LIN {X 0,Y 281.537,Z 487.928,A -85,B 0,C 180,E1 -17516.689,E2 -17516.689} C_VEL
LIN {X 0,Y 281.333,Z 491.576,A -85,B 0,C 180,E1 -17518.052,E2 -17518.052} C_VEL
LIN {X 0,Y 285.942,Z 506.962,A -85,B 0,C 180,E1 -17519.189,E2 -17519.189} C_VEL
LIN {X 0,Y 289.242,Z 521.138,A -85,B 0,C 180,E1 -17520.411,E2 -17520.411} C_VEL
LIN {X 0,Y 291.221,Z 533.956,A -85,B 0,C 180,E1 -17521.672,E2 -17521.672} C_VEL
LIN {X 0,Y 291.985,Z 542.885,A -85,B 0,C 180,E1 -17522.647,E2 -17522.647} C_VEL
LIN {X 0,Y 290.191,Z 554.779,A -85,B 0,C 180,E1 -17523.912,E2 -17523.912} C_VEL
LIN {X 0,Y 287.889,Z 566.73,A -85,B 0,C 180,E1 -17525.48,E2 -17525.48} C_VEL
LIN {X 0,Y 285.539,Z 577.345,A -85,B 0,C 180,E1 -17527.191,E2 -17527.191} C_VEL
LIN {X 0,Y 283.172,Z 587.851,A -85,B 0,C 180,E1 -17529.288,E2 -17529.288} C_VEL
LIN {X 0,Y 281.044,Z 596.524,A -85,B 0,C 180,E1 -17531.408,E2 -17531.408} C_VEL
LIN {X 0,Y 279.492,Z 603.728,A -85,B 0,C 180,E1 -17533.567,E2 -17533.567} C_VEL
LIN {X 0,Y 277.872,Z 610.612,A -85,B 0,C 180,E1 -17536.097,E2 -17536.097} C_VEL
LIN {X 0,Y 276.558,Z 616.782,A -85,B 0,C 180,E1 -17539.013,E2 -17539.013} C_VEL
LIN {X 0,Y 275.927,Z 620.289,A -85,B 0,C 180,E1 -17541.209,E2 -17541.209} C_VEL
LIN {X 0,Y 275.417,Z 623.71,A -85,B 0,C 180,E1 -17544.142,E2 -17544.142} C_VEL
LIN {X 0,Y 275.26,Z 625.741,A -85,B 0,C 180,E1 -17547.073,E2 -17547.073} C_VEL
LIN {X 0,Y 275.22,Z 626.437,A -85,B 0,C 180,E1 -17550,E2 -17550} C_VEL
LIN {X 0,Y 275.258,Z 625.8,A -85,B 0,C 180,E1 -17552.927,E2 -17552.927} C_VEL
LIN {X 0,Y 275.416,Z 623.816,A -85,B 0,C 180,E1 -17555.858,E2 -17555.858} C_VEL
LIN {X 0,Y 275.925,Z 620.448,A -85,B 0,C 180,E1 -17558.791,E2 -17558.791} C_VEL
LIN {X 0,Y 276.784,Z 615.594,A -85,B 0,C 180,E1 -17561.72,E2 -17561.72} C_VEL
LIN {X 0,Y 277.821,Z 610.887,A -85,B 0,C 180,E1 -17563.905,E2 -17563.905} C_VEL
LIN {X 0,Y 279.41,Z 604.105,A -85,B 0,C 180,E1 -17566.423,E2 -17566.423} C_VEL
LIN {X 0,Y 281.359,Z 595.594,A -85,B 0,C 180,E1 -17568.949,E2 -17568.949} C_VEL
LIN {X 0,Y 283.505,Z 586.735,A -85,B 0,C 180,E1 -17571.067,E2 -17571.067} C_VEL
LIN {X 0,Y 285.86,Z 576.009,A -85,B 0,C 180,E1 -17573.164,E2 -17573.164} C_VEL
LIN {X 0,Y 288.304,Z 565.121,A -85,B 0,C 180,E1 -17574.866,E2 -17574.866} C_VEL
LIN {X 0,Y 290.592,Z 552.488,A -85,B 0,C 180,E1 -17576.467,E2 -17576.467} C_VEL
LIN {X 0,Y 292.06,Z 542.514,A -85,B 0,C 180,E1 -17577.505,E2 -17577.505} C_VEL
LIN {X 0,Y 290.791,Z 530.649,A -85,B 0,C 180,E1 -17578.792,E2 -17578.792} C_VEL
LIN {X 0,Y 288.442,Z 517.113,A -85,B 0,C 180,E1 -17580.077,E2 -17580.077} C_VEL
LIN {X 0,Y 284.962,Z 503.246,A -85,B 0,C 180,E1 -17581.223,E2 -17581.223} C_VEL
LIN {X 0,Y 281.275,Z 491.314,A -85,B 0,C 180,E1 -17582.094,E2 -17582.094} C_VEL
LIN {X 0,Y 282.191,Z 480.989,A -85,B 0,C 180,E1 -17586.263,E2 -17586.263} C_VEL
LIN {X 0,Y 283.218,Z 471.628,A -85,B 0,C 180,E1 -17590.18,E2 -17590.18} C_VEL
LIN {X 0,Y 283.249,Z 467.404,A -85,B 0,C 180,E1 -17592.061,E2 -17592.061} C_VEL
LIN {X 0,Y 281.982,Z 459.837,A -85,B 0,C 180,E1 -17595.744,E2 -17595.744} C_VEL
LIN {X 0,Y 280.547,Z 452.755,A -85,B 0,C 180,E1 -17599.358,E2 -17599.358} C_VEL
LIN {X 0,Y 279.094,Z 446.242,A -85,B 0,C 180,E1 -17602.817,E2 -17602.817} C_VEL
LIN {X 0,Y 277.267,Z 439.563,A -85,B 0,C 180,E1 -17606.638,E2 -17606.638} C_VEL
LIN {X 0,Y 277.277,Z 439.557,A -85,B 0,C 180,E1 -17609.73,E2 -17609.73} C_VEL
LIN {X 0,Y 282.338,Z 455.073,A -85,B 0,C 180,E1 -17611.505,E2 -17611.505} C_VEL
LIN {X 0,Y 286.61,Z 469.194,A -85,B 0,C 180,E1 -17613.343,E2 -17613.343} C_VEL
LIN {X 0,Y 287.766,Z 473.23,A -85,B 0,C 180,E1 -17613.921,E2 -17613.921} C_VEL
LIN {X 0,Y 286.168,Z 485.511,A -85,B 0,C 180,E1 -17615.516,E2 -17615.516} C_VEL
LIN {X 0,Y 284.267,Z 498.156,A -85,B 0,C 180,E1 -17617.467,E2 -17617.467} C_VEL
LIN {X 0,Y 282.497,Z 509.782,A -85,B 0,C 180,E1 -17619.617,E2 -17619.617} C_VEL
LIN {X 0,Y 280.89,Z 519.521,A -85,B 0,C 180,E1 -17621.752,E2 -17621.752} C_VEL
LIN {X 0,Y 279.534,Z 529.33,A -85,B 0,C 180,E1 -17624.319,E2 -17624.319} C_VEL
LIN {X 0,Y 279.286,Z 530.981,A -85,B 0,C 180,E1 -17624.798,E2 -17624.798} C_VEL
LIN {X 0,Y 278.057,Z 534.299,A -85,B 0,C 180,E1 -17625.786,E2 -17625.786} C_VEL
LIN {X 0,Y 274.501,Z 539.379,A -85,B 0,C 180,E1 -17627.397,E2 -17627.397} C_VEL
LIN {X 0,Y 271.128,Z 544.003,A -85,B 0,C 180,E1 -17629.093,E2 -17629.093} C_VEL
LIN {X 0,Y 270.198,Z 546.576,A -85,B 0,C 180,E1 -17630.195,E2 -17630.195} C_VEL
LIN {X 0,Y 269.657,Z 552.512,A -85,B 0,C 180,E1 -17633.265,E2 -17633.265} C_VEL
LIN {X 0,Y 269.565,Z 555.917,A -85,B 0,C 180,E1 -17635.514,E2 -17635.514} C_VEL
LIN {X 0,Y 269.279,Z 559.358,A -85,B 0,C 180,E1 -17638.504,E2 -17638.504} C_VEL
LIN {X 0,Y 269.373,Z 561.559,A -85,B 0,C 180,E1 -17641.495,E2 -17641.495} C_VEL
LIN {X 0,Y 269.987,Z 562.568,A -85,B 0,C 180,E1 -17644.479,E2 -17644.479} C_VEL
LIN {X 0,Y 271.059,Z 562.393,A -85,B 0,C 180,E1 -17647.449,E2 -17647.449} C_VEL
LIN {X 0,Y 272.422,Z 561.092,A -85,B 0,C 180,E1 -17650.404,E2 -17650.404} C_VEL
LIN {X 0,Y 274.151,Z 558.636,A -85,B 0,C 180,E1 -17653.339,E2 -17653.339} C_VEL
LIN {X 0,Y 276.346,Z 555.017,A -85,B 0,C 180,E1 -17656.245,E2 -17656.245} C_VEL
LIN {X 0,Y 279.276,Z 550.056,A -85,B 0,C 180,E1 -17659.096,E2 -17659.096} C_VEL
LIN {X 0,Y 281.817,Z 545.44,A -85,B 0,C 180,E1 -17661.199,E2 -17661.199} C_VEL
LIN {X 0,Y 286.188,Z 537.267,A -85,B 0,C 180,E1 -17664.197,E2 -17664.197} C_VEL
LIN {X 0,Y 290.835,Z 527.733,A -85,B 0,C 180,E1 -17666.942,E2 -17666.942} C_VEL
LIN {X 0,Y 295.354,Z 517.993,A -85,B 0,C 180,E1 -17669.196,E2 -17669.196} C_VEL
LIN {X 0,Y 299.707,Z 508.242,A -85,B 0,C 180,E1 -17671.057,E2 -17671.057} C_VEL
LIN {X 0,Y 303.199,Z 499.743,A -85,B 0,C 180,E1 -17672.464,E2 -17672.464} C_VEL
LIN {X 0,Y 303.462,Z 498.058,A -85,B 0,C 180,E1 -17672.86,E2 -17672.86} C_VEL
LIN {X 0,Y 302.842,Z 492.133,A -85,B 0,C 180,E1 -17674.941,E2 -17674.941} C_VEL
LIN {X 0,Y 302.211,Z 488.957,A -85,B 0,C 180,E1 -17676.323,E2 -17676.323} C_VEL
LIN {X 0,Y 301.253,Z 487.359,A -85,B 0,C 180,E1 -17677.515,E2 -17677.515} C_VEL
LIN {X 0,Y 299.735,Z 486.025,A -85,B 0,C 180,E1 -17679.307,E2 -17679.307} C_VEL
LIN {X 0,Y 298.35,Z 485.722,A -85,B 0,C 180,E1 -17681.267,E2 -17681.267} C_VEL
LIN {X 0,Y 297.068,Z 486.886,A -85,B 0,C 180,E1 -17683.32,E2 -17683.32} C_VEL
LIN {X 0,Y 296.328,Z 488.596,A -85,B 0,C 180,E1 -17684.642,E2 -17684.642} C_VEL
LIN {X 0,Y 294.815,Z 495.196,A -85,B 0,C 180,E1 -17687.646,E2 -17687.646} C_VEL
LIN {X 0,Y 294.665,Z 498.561,A -85,B 0,C 180,E1 -17689.057,E2 -17689.057} C_VEL
LIN {X 0,Y 294.316,Z 505.488,A -85,B 0,C 180,E1 -17691.235,E2 -17691.235} C_VEL
LIN {X 0,Y 294.003,Z 512.7,A -85,B 0,C 180,E1 -17693.139,E2 -17693.139} C_VEL
LIN {X 0,Y 293.508,Z 520.438,A -85,B 0,C 180,E1 -17694.923,E2 -17694.923} C_VEL
LIN {X 0,Y 292.34,Z 530.113,A -85,B 0,C 180,E1 -17696.885,E2 -17696.885} C_VEL
LIN {X 0,Y 290.404,Z 539.351,A -85,B 0,C 180,E1 -17698.604,E2 -17698.604} C_VEL
LIN {X 0,Y 287.008,Z 552.38,A -85,B 0,C 180,E1 -17701.078,E2 -17701.078} C_VEL
LIN {X 0,Y 285.923,Z 557.42,A -85,B 0,C 180,E1 -17702.159,E2 -17702.159} C_VEL
LIN {X 0,Y 282.042,Z 567.163,A -85,B 0,C 180,E1 -17704.147,E2 -17704.147} C_VEL
LIN {X 0,Y 281.188,Z 569.389,A -85,B 0,C 180,E1 -17704.658,E2 -17704.658} C_VEL
LIN {X 0,Y 278.988,Z 579.397,A -85,B 0,C 180,E1 -17706.231,E2 -17706.231} C_VEL
LIN {X 0,Y 276.824,Z 588.72,A -85,B 0,C 180,E1 -17708.008,E2 -17708.008} C_VEL
LIN {X 0,Y 274.587,Z 598.075,A -85,B 0,C 180,E1 -17710.176,E2 -17710.176} C_VEL
LIN {X 0,Y 272.687,Z 606.145,A -85,B 0,C 180,E1 -17712.479,E2 -17712.479} C_VEL
LIN {X 0,Y 271.131,Z 613.215,A -85,B 0,C 180,E1 -17714.977,E2 -17714.977} C_VEL
LIN {X 0,Y 269.555,Z 619.823,A -85,B 0,C 180,E1 -17717.961,E2 -17717.961} C_VEL
LIN {X 0,Y 268.738,Z 624.77,A -85,B 0,C 180,E1 -17720.972,E2 -17720.972} C_VEL
LIN {X 0,Y 268.305,Z 628.21,A -85,B 0,C 180,E1 -17723.986,E2 -17723.986} C_VEL
LIN {X 0,Y 268.201,Z 630.245,A -85,B 0,C 180,E1 -17726.996,E2 -17726.996} C_VEL
LIN {X 0,Y 268.193,Z 630.919,A -85,B 0,C 180,E1 -17730,E2 -17730} C_VEL
LIN {X 0,Y 268.199,Z 630.236,A -85,B 0,C 180,E1 -17733.004,E2 -17733.004} C_VEL
LIN {X 0,Y 268.299,Z 628.194,A -85,B 0,C 180,E1 -17736.014,E2 -17736.014} C_VEL
LIN {X 0,Y 268.714,Z 624.745,A -85,B 0,C 180,E1 -17739.028,E2 -17739.028} C_VEL
LIN {X 0,Y 269.537,Z 619.783,A -85,B 0,C 180,E1 -17742.04,E2 -17742.04} C_VEL
LIN {X 0,Y 271.095,Z 613.165,A -85,B 0,C 180,E1 -17745.025,E2 -17745.025} C_VEL
LIN {X 0,Y 272.585,Z 606.058,A -85,B 0,C 180,E1 -17747.535,E2 -17747.535} C_VEL
LIN {X 0,Y 274.558,Z 597.994,A -85,B 0,C 180,E1 -17749.826,E2 -17749.826} C_VEL
LIN {X 0,Y 276.769,Z 588.618,A -85,B 0,C 180,E1 -17751.996,E2 -17751.996} C_VEL
LIN {X 0,Y 279.183,Z 578.215,A -85,B 0,C 180,E1 -17753.949,E2 -17753.949} C_VEL
LIN {X 0,Y 281.738,Z 566.352,A -85,B 0,C 180,E1 -17755.741,E2 -17755.741} C_VEL
LIN {X 0,Y 283.764,Z 553.932,A -85,B 0,C 180,E1 -17757.27,E2 -17757.27} C_VEL
LIN {X 0,Y 283.178,Z 541.327,A -85,B 0,C 180,E1 -17758.748,E2 -17758.748} C_VEL
LIN {X 0,Y 281.859,Z 528.409,A -85,B 0,C 180,E1 -17760.039,E2 -17760.039} C_VEL
LIN {X 0,Y 280.013,Z 514.186,A -85,B 0,C 180,E1 -17761.189,E2 -17761.189} C_VEL
LIN {X 0,Y 277.183,Z 503.097,A -85,B 0,C 180,E1 -17762.029,E2 -17762.029} C_VEL
LIN {X 0,Y 272.899,Z 489.832,A -85,B 0,C 180,E1 -17763.066,E2 -17763.066} C_VEL
LIN {X 0,Y 271.754,Z 479.976,A -85,B 0,C 180,E1 -17765.129,E2 -17765.129} C_VEL
LIN {X 0,Y 270.998,Z 474.249,A -85,B 0,C 180,E1 -17766.39,E2 -17766.39} C_VEL
LIN {X 0,Y 271.661,Z 468.446,A -85,B 0,C 180,E1 -17770.298,E2 -17770.298} C_VEL
LIN {X 0,Y 272.367,Z 462.83,A -85,B 0,C 180,E1 -17774.162,E2 -17774.162} C_VEL
LIN {X 0,Y 272.893,Z 458.634,A -85,B 0,C 180,E1 -17777.089,E2 -17777.089} C_VEL
LIN {X 0,Y 272.752,Z 454.791,A -85,B 0,C 180,E1 -17779.896,E2 -17779.896} C_VEL
LIN {X 0,Y 271.911,Z 450.029,A -85,B 0,C 180,E1 -17783.525,E2 -17783.525} C_VEL
LIN {X 0,Y 271.032,Z 444.568,A -85,B 0,C 180,E1 -17787.888,E2 -17787.888} C_VEL
LIN {X 0,Y 270.308,Z 440.441,A -85,B 0,C 180,E1 -17791.462,E2 -17791.462} C_VEL
LIN {X 0,Y 270.278,Z 440.435,A -85,B 0,C 180,E1 -17795.519,E2 -17795.519} C_VEL
LIN {X 0,Y 270.303,Z 440.421,A -85,B 0,C 180,E1 -17800.245,E2 -17800.245} C_VEL
LIN {X 0,Y 270.404,Z 440.405,A -85,B 0,C 180,E1 -17804.936,E2 -17804.936} C_VEL
LIN {X 0,Y 270.411,Z 440.415,A -85,B 0,C 180,E1 -17809.518,E2 -17809.518} C_VEL
LIN {X 0,Y 270.582,Z 440.392,A -85,B 0,C 180,E1 -17812.538,E2 -17812.538} C_VEL
LIN {X 0,Y 270.789,Z 440.366,A -85,B 0,C 180,E1 -17818.513,E2 -17818.513} C_VEL
LIN {X 0,Y 270.789,Z 440.369,A -85,B 0,C 180,E1 -17821.487,E2 -17821.487} C_VEL
LIN {X 0,Y 270.613,Z 440.387,A -85,B 0,C 180,E1 -17827.461,E2 -17827.461} C_VEL
LIN {X 0,Y 270.444,Z 440.419,A -85,B 0,C 180,E1 -17830.481,E2 -17830.481} C_VEL
LIN {X 0,Y 270.405,Z 440.418,A -85,B 0,C 180,E1 -17835.065,E2 -17835.065} C_VEL
LIN {X 0,Y 270.301,Z 440.432,A -85,B 0,C 180,E1 -17839.756,E2 -17839.756} C_VEL
LIN {X 0,Y 270.239,Z 440.448,A -85,B 0,C 180,E1 -17844.589,E2 -17844.589} C_VEL
LIN {X 0,Y 270.273,Z 440.44,A -85,B 0,C 180,E1 -17847.909,E2 -17847.909} C_VEL
LIN {X 0,Y 270.237,Z 440.596,A -85,B 0,C 180,E1 -17852.438,E2 -17852.438} C_VEL
LIN {X 0,Y 271.699,Z 445.957,A -85,B 0,C 180,E1 -17855.592,E2 -17855.592} C_VEL
LIN {X 0,Y 273.306,Z 452.497,A -85,B 0,C 180,E1 -17859.194,E2 -17859.194} C_VEL
LIN {X 0,Y 274.734,Z 459,A -85,B 0,C 180,E1 -17862.679,E2 -17862.679} C_VEL
LIN {X 0,Y 276.105,Z 466.777,A -85,B 0,C 180,E1 -17866.586,E2 -17866.586} C_VEL
LIN {X 0,Y 276.618,Z 471.079,A -85,B 0,C 180,E1 -17868.656,E2 -17868.656} C_VEL
LIN {X 0,Y 275.952,Z 477.382,A -85,B 0,C 180,E1 -17871.394,E2 -17871.394} C_VEL
LIN {X 0,Y 274.979,Z 486.758,A -85,B 0,C 180,E1 -17875.306,E2 -17875.306} C_VEL
LIN {X 0,Y 274.573,Z 491.348,A -85,B 0,C 180,E1 -17877.163,E2 -17877.163} C_VEL
LIN {X 0,Y 279.426,Z 507.204,A -85,B 0,C 180,E1 -17878.401,E2 -17878.401} C_VEL
LIN {X 0,Y 282.623,Z 521.049,A -85,B 0,C 180,E1 -17879.638,E2 -17879.638} C_VEL
LIN {X 0,Y 284.651,Z 533.995,A -85,B 0,C 180,E1 -17880.956,E2 -17880.956} C_VEL
LIN {X 0,Y 285.511,Z 544.157,A -85,B 0,C 180,E1 -17882.115,E2 -17882.115} C_VEL
LIN {X 0,Y 283.482,Z 556.585,A -85,B 0,C 180,E1 -17883.497,E2 -17883.497} C_VEL
LIN {X 0,Y 281.179,Z 567.932,A -85,B 0,C 180,E1 -17885.053,E2 -17885.053} C_VEL
LIN {X 0,Y 278.967,Z 577.399,A -85,B 0,C 180,E1 -17886.622,E2 -17886.622} C_VEL
LIN {X 0,Y 276.535,Z 587.906,A -85,B 0,C 180,E1 -17888.767,E2 -17888.767} C_VEL
LIN {X 0,Y 274.293,Z 596.579,A -85,B 0,C 180,E1 -17890.932,E2 -17890.932} C_VEL
LIN {X 0,Y 272.609,Z 603.855,A -85,B 0,C 180,E1 -17893.164,E2 -17893.164} C_VEL
LIN {X 0,Y 271.448,Z 608.885,A -85,B 0,C 180,E1 -17894.995,E2 -17894.995} C_VEL
LIN {X 0,Y 270.171,Z 613.968,A -85,B 0,C 180,E1 -17897.226,E2 -17897.226} C_VEL
LIN {X 0,Y 269.072,Z 619.296,A -85,B 0,C 180,E1 -17900.225,E2 -17900.225} C_VEL
LIN {X 0,Y 268.56,Z 622.238,A -85,B 0,C 180,E1 -17902.482,E2 -17902.482} C_VEL
LIN {X 0,Y 268.203,Z 624.954,A -85,B 0,C 180,E1 -17905.491,E2 -17905.491} C_VEL
LIN {X 0,Y 268.141,Z 626.313,A -85,B 0,C 180,E1 -17908.498,E2 -17908.498} C_VEL
LIN {X 0,Y 268.14,Z 626.344,A -85,B 0,C 180,E1 -17911.502,E2 -17911.502} C_VEL
LIN {X 0,Y 268.198,Z 625.035,A -85,B 0,C 180,E1 -17914.509,E2 -17914.509} C_VEL
LIN {X 0,Y 268.549,Z 622.368,A -85,B 0,C 180,E1 -17917.519,E2 -17917.519} C_VEL
LIN {X 0,Y 269.276,Z 618.272,A -85,B 0,C 180,E1 -17920.527,E2 -17920.527} C_VEL
LIN {X 0,Y 270.443,Z 612.62,A -85,B 0,C 180,E1 -17923.526,E2 -17923.526} C_VEL
LIN {X 0,Y 272.169,Z 606.227,A -85,B 0,C 180,E1 -17926.116,E2 -17926.116} C_VEL
LIN {X 0,Y 273.991,Z 598.286,A -85,B 0,C 180,E1 -17928.701,E2 -17928.701} C_VEL
LIN {X 0,Y 276.058,Z 589.958,A -85,B 0,C 180,E1 -17930.88,E2 -17930.88} C_VEL
LIN {X 0,Y 278.468,Z 579.891,A -85,B 0,C 180,E1 -17933.029,E2 -17933.029} C_VEL
LIN {X 0,Y 281.049,Z 568.621,A -85,B 0,C 180,E1 -17934.96,E2 -17934.96} C_VEL
LIN {X 0,Y 283.378,Z 557.414,A -85,B 0,C 180,E1 -17936.514,E2 -17936.514} C_VEL
LIN {X 0,Y 285.598,Z 543.959,A -85,B 0,C 180,E1 -17938.017,E2 -17938.017} C_VEL
LIN {X 0,Y 284.481,Z 532.457,A -85,B 0,C 180,E1 -17939.326,E2 -17939.326} C_VEL
LIN {X 0,Y 282.182,Z 518.597,A -85,B 0,C 180,E1 -17940.71,E2 -17940.71} C_VEL
LIN {X 0,Y 279.027,Z 505.702,A -85,B 0,C 180,E1 -17941.847,E2 -17941.847} C_VEL
LIN {X 0,Y 274.583,Z 491.242,A -85,B 0,C 180,E1 -17943.003,E2 -17943.003} C_VEL
LIN {X 0,Y 275.604,Z 480.868,A -85,B 0,C 180,E1 -17947.274,E2 -17947.274} C_VEL
LIN {X 0,Y 276.534,Z 472.831,A -85,B 0,C 180,E1 -17950.697,E2 -17950.697} C_VEL
LIN {X 0,Y 276.43,Z 468.936,A -85,B 0,C 180,E1 -17952.498,E2 -17952.498} C_VEL
LIN {X 0,Y 275.429,Z 462.706,A -85,B 0,C 180,E1 -17955.599,E2 -17955.599} C_VEL
LIN {X 0,Y 274.056,Z 455.847,A -85,B 0,C 180,E1 -17959.161,E2 -17959.161} C_VEL
LIN {X 0,Y 272.431,Z 448.564,A -85,B 0,C 180,E1 -17963.103,E2 -17963.103} C_VEL
LIN {X 0,Y 270.575,Z 441.975,A -85,B 0,C 180,E1 -17966.944,E2 -17966.944} C_VEL
LIN {X 0,Y 270.198,Z 440.454,A -85,B 0,C 180,E1 -17967.887,E2 -17967.887} C_VEL
LIN {X 0,Y 270.208,Z 440.438,A -85,B 0,C 180,E1 -17969.262,E2 -17969.262} C_VEL
LIN {X 0,Y 274.919,Z 454.754,A -85,B 0,C 180,E1 -17970.941,E2 -17970.941} C_VEL
LIN {X 0,Y 278.914,Z 467.876,A -85,B 0,C 180,E1 -17972.678,E2 -17972.678} C_VEL
LIN {X 0,Y 280.801,Z 474.405,A -85,B 0,C 180,E1 -17973.624,E2 -17973.624} C_VEL
LIN {X 0,Y 280.034,Z 481.499,A -85,B 0,C 180,E1 -17974.546,E2 -17974.546} C_VEL
LIN {X 0,Y 277.986,Z 494.946,A -85,B 0,C 180,E1 -17976.535,E2 -17976.535} C_VEL
LIN {X 0,Y 276.04,Z 507.187,A -85,B 0,C 180,E1 -17978.727,E2 -17978.727} C_VEL
LIN {X 0,Y 274.271,Z 517.708,A -85,B 0,C 180,E1 -17980.969,E2 -17980.969} C_VEL
LIN {X 0,Y 272.99,Z 526.414,A -85,B 0,C 180,E1 -17983.164,E2 -17983.164} C_VEL
LIN {X 0,Y 271.638,Z 535.137,A -85,B 0,C 180,E1 -17985.771,E2 -17985.771} C_VEL
LIN {X 0,Y 270.592,Z 543.292,A -85,B 0,C 180,E1 -17988.767,E2 -17988.767} C_VEL
LIN {X 0,Y 270.198,Z 546.576,A -85,B 0,C 180,E1 -17990.195,E2 -17990.195} C_VEL
LIN {X 0,Y 269.313,Z 549.046,A -85,B 0,C 180,E1 -17991.317,E2 -17991.317} C_VEL
LIN {X 0,Y 266.197,Z 552.693,A -85,B 0,C 180,E1 -17993.173,E2 -17993.173} C_VEL
LIN {X 0,Y 263.622,Z 555.289,A -85,B 0,C 180,E1 -17994.712,E2 -17994.712} C_VEL
LIN {X 0,Y 262.475,Z 557.024,A -85,B 0,C 180,E1 -17995.927,E2 -17995.927} C_VEL
LIN {X 0,Y 262.353,Z 557.506,A -85,B 0,C 180,E1 -17996.342,E2 -17996.342} C_VEL
LIN {X 0,Y 262.213,Z 559.894,A -85,B 0,C 180,E1 -17998.464,E2 -17998.464} C_VEL
LIN {X 0,Y 262.337,Z 562.272,A -85,B 0,C 180,E1 -18001.535,E2 -18001.535} C_VEL
LIN {X 0,Y 262.976,Z 563.458,A -85,B 0,C 180,E1 -18004.598,E2 -18004.598} C_VEL
LIN {X 0,Y 264.1,Z 563.469,A -85,B 0,C 180,E1 -18007.646,E2 -18007.646} C_VEL
LIN {X 0,Y 265.553,Z 562.332,A -85,B 0,C 180,E1 -18010.676,E2 -18010.676} C_VEL
LIN {X 0,Y 267.384,Z 560.076,A -85,B 0,C 180,E1 -18013.683,E2 -18013.683} C_VEL
LIN {X 0,Y 269.739,Z 556.631,A -85,B 0,C 180,E1 -18016.655,E2 -18016.655} C_VEL
LIN {X 0,Y 272.825,Z 551.933,A -85,B 0,C 180,E1 -18019.565,E2 -18019.565} C_VEL
LIN {X 0,Y 276.545,Z 545.91,A -85,B 0,C 180,E1 -18022.408,E2 -18022.408} C_VEL
LIN {X 0,Y 280.84,Z 538.447,A -85,B 0,C 180,E1 -18025.177,E2 -18025.177} C_VEL
LIN {X 0,Y 284.893,Z 530.882,A -85,B 0,C 180,E1 -18027.471,E2 -18027.471} C_VEL
LIN {X 0,Y 289.778,Z 521.41,A -85,B 0,C 180,E1 -18029.814,E2 -18029.814} C_VEL
LIN {X 0,Y 295.091,Z 510.429,A -85,B 0,C 180,E1 -18032,E2 -18032} C_VEL
LIN {X 0,Y 298.137,Z 503.586,A -85,B 0,C 180,E1 -18033.177,E2 -18033.177} C_VEL
LIN {X 0,Y 298.598,Z 502.215,A -85,B 0,C 180,E1 -18033.465,E2 -18033.465} C_VEL
LIN {X 0,Y 298.353,Z 496.969,A -85,B 0,C 180,E1 -18035.455,E2 -18035.455} C_VEL
LIN {X 0,Y 297.962,Z 494.409,A -85,B 0,C 180,E1 -18036.683,E2 -18036.683} C_VEL
LIN {X 0,Y 296.547,Z 492.579,A -85,B 0,C 180,E1 -18038.548,E2 -18038.548} C_VEL
LIN {X 0,Y 295.293,Z 491.93,A -85,B 0,C 180,E1 -18040.394,E2 -18040.394} C_VEL
LIN {X 0,Y 294.158,Z 492.361,A -85,B 0,C 180,E1 -18042.213,E2 -18042.213} C_VEL
LIN {X 0,Y 292.969,Z 494.251,A -85,B 0,C 180,E1 -18044.081,E2 -18044.081} C_VEL
LIN {X 0,Y 291.354,Z 498.927,A -85,B 0,C 180,E1 -18046.357,E2 -18046.357} C_VEL
LIN {X 0,Y 290.675,Z 503.868,A -85,B 0,C 180,E1 -18048.549,E2 -18048.549} C_VEL
LIN {X 0,Y 289.863,Z 511.203,A -85,B 0,C 180,E1 -18050.921,E2 -18050.921} C_VEL
LIN {X 0,Y 289.105,Z 518.87,A -85,B 0,C 180,E1 -18053.005,E2 -18053.005} C_VEL
LIN {X 0,Y 288.002,Z 527.223,A -85,B 0,C 180,E1 -18054.952,E2 -18054.952} C_VEL
LIN {X 0,Y 286.309,Z 535.869,A -85,B 0,C 180,E1 -18056.751,E2 -18056.751} C_VEL
LIN {X 0,Y 283.557,Z 545.561,A -85,B 0,C 180,E1 -18058.635,E2 -18058.635} C_VEL
LIN {X 0,Y 280.576,Z 555.757,A -85,B 0,C 180,E1 -18060.762,E2 -18060.762} C_VEL
LIN {X 0,Y 279.796,Z 558.934,A -85,B 0,C 180,E1 -18061.494,E2 -18061.494} C_VEL
LIN {X 0,Y 275.141,Z 569.677,A -85,B 0,C 180,E1 -18063.856,E2 -18063.856} C_VEL
LIN {X 0,Y 274.123,Z 572.267,A -85,B 0,C 180,E1 -18064.466,E2 -18064.466} C_VEL
LIN {X 0,Y 271.54,Z 583.248,A -85,B 0,C 180,E1 -18066.349,E2 -18066.349} C_VEL
LIN {X 0,Y 269.025,Z 593.574,A -85,B 0,C 180,E1 -18068.547,E2 -18068.547} C_VEL
LIN {X 0,Y 266.837,Z 602.075,A -85,B 0,C 180,E1 -18070.778,E2 -18070.778} C_VEL
LIN {X 0,Y 264.918,Z 610.174,A -85,B 0,C 180,E1 -18073.43,E2 -18073.43} C_VEL
LIN {X 0,Y 263.335,Z 616.682,A -85,B 0,C 180,E1 -18076.102,E2 -18076.102} C_VEL
LIN {X 0,Y 262.073,Z 622.437,A -85,B 0,C 180,E1 -18079.18,E2 -18079.18} C_VEL
LIN {X 0,Y 261.4,Z 626.613,A -85,B 0,C 180,E1 -18082.274,E2 -18082.274} C_VEL
LIN {X 0,Y 261.105,Z 629.34,A -85,B 0,C 180,E1 -18085.368,E2 -18085.368} C_VEL
LIN {X 0,Y 261.115,Z 630.694,A -85,B 0,C 180,E1 -18088.458,E2 -18088.458} C_VEL
LIN {X 0,Y 261.114,Z 630.689,A -85,B 0,C 180,E1 -18091.542,E2 -18091.542} C_VEL
LIN {X 0,Y 261.1,Z 629.328,A -85,B 0,C 180,E1 -18094.632,E2 -18094.632} C_VEL
LIN {X 0,Y 261.374,Z 626.592,A -85,B 0,C 180,E1 -18097.726,E2 -18097.726} C_VEL
LIN {X 0,Y 262.062,Z 622.402,A -85,B 0,C 180,E1 -18100.82,E2 -18100.82} C_VEL
LIN {X 0,Y 263.318,Z 616.634,A -85,B 0,C 180,E1 -18103.899,E2 -18103.899} C_VEL
LIN {X 0,Y 264.855,Z 610.115,A -85,B 0,C 180,E1 -18106.574,E2 -18106.574} C_VEL
LIN {X 0,Y 266.801,Z 601.997,A -85,B 0,C 180,E1 -18109.225,E2 -18109.225} C_VEL
LIN {X 0,Y 268.959,Z 593.478,A -85,B 0,C 180,E1 -18111.458,E2 -18111.458} C_VEL
LIN {X 0,Y 271.483,Z 583.129,A -85,B 0,C 180,E1 -18113.657,E2 -18113.657} C_VEL
LIN {X 0,Y 273.937,Z 572.705,A -85,B 0,C 180,E1 -18115.451,E2 -18115.451} C_VEL
LIN {X 0,Y 276.333,Z 560.88,A -85,B 0,C 180,E1 -18117.107,E2 -18117.107} C_VEL
LIN {X 0,Y 277.245,Z 555.459,A -85,B 0,C 180,E1 -18117.762,E2 -18117.762} C_VEL
LIN {X 0,Y 276.823,Z 543.248,A -85,B 0,C 180,E1 -18119.265,E2 -18119.265} C_VEL
LIN {X 0,Y 275.638,Z 529.952,A -85,B 0,C 180,E1 -18120.66,E2 -18120.66} C_VEL
LIN {X 0,Y 273.849,Z 515.447,A -85,B 0,C 180,E1 -18121.897,E2 -18121.897} C_VEL
LIN {X 0,Y 270.615,Z 503.053,A -85,B 0,C 180,E1 -18122.905,E2 -18122.905} C_VEL
LIN {X 0,Y 266.326,Z 489.897,A -85,B 0,C 180,E1 -18123.992,E2 -18123.992} C_VEL
LIN {X 0,Y 264.705,Z 476.756,A -85,B 0,C 180,E1 -18126.914,E2 -18126.914} C_VEL
LIN {X 0,Y 264.168,Z 472.303,A -85,B 0,C 180,E1 -18127.968,E2 -18127.968} C_VEL
LIN {X 0,Y 265.024,Z 465.481,A -85,B 0,C 180,E1 -18132.722,E2 -18132.722} C_VEL
LIN {X 0,Y 265.747,Z 460.1,A -85,B 0,C 180,E1 -18136.559,E2 -18136.559} C_VEL
LIN {X 0,Y 265.857,Z 457.291,A -85,B 0,C 180,E1 -18138.633,E2 -18138.633} C_VEL
LIN {X 0,Y 265.361,Z 453.495,A -85,B 0,C 180,E1 -18141.509,E2 -18141.509} C_VEL
LIN {X 0,Y 264.327,Z 447.802,A -85,B 0,C 180,E1 -18146.058,E2 -18146.058} C_VEL
LIN {X 0,Y 263.643,Z 443.575,A -85,B 0,C 180,E1 -18149.57,E2 -18149.57} C_VEL
LIN {X 0,Y 263.276,Z 441.316,A -85,B 0,C 180,E1 -18151.598,E2 -18151.598} C_VEL
LIN {X 0,Y 263.227,Z 441.308,A -85,B 0,C 180,E1 -18155.2,E2 -18155.2} C_VEL
LIN {X 0,Y 263.265,Z 441.295,A -85,B 0,C 180,E1 -18159.694,E2 -18159.694} C_VEL
LIN {X 0,Y 263.352,Z 441.284,A -85,B 0,C 180,E1 -18164.522,E2 -18164.522} C_VEL
LIN {X 0,Y 263.354,Z 441.298,A -85,B 0,C 180,E1 -18169.234,E2 -18169.234} C_VEL
LIN {X 0,Y 263.542,Z 441.266,A -85,B 0,C 180,E1 -18172.338,E2 -18172.338} C_VEL
LIN {X 0,Y 263.753,Z 441.241,A -85,B 0,C 180,E1 -18178.473,E2 -18178.473} C_VEL
LIN {X 0,Y 263.753,Z 441.244,A -85,B 0,C 180,E1 -18181.527,E2 -18181.527} C_VEL
LIN {X 0,Y 263.575,Z 441.261,A -85,B 0,C 180,E1 -18187.662,E2 -18187.662} C_VEL
LIN {X 0,Y 263.376,Z 441.302,A -85,B 0,C 180,E1 -18190.766,E2 -18190.766} C_VEL
LIN {X 0,Y 263.352,Z 441.302,A -85,B 0,C 180,E1 -18195.478,E2 -18195.478} C_VEL
LIN {X 0,Y 263.264,Z 441.316,A -85,B 0,C 180,E1 -18200.307,E2 -18200.307} C_VEL
LIN {X 0,Y 263.195,Z 441.324,A -85,B 0,C 180,E1 -18205.293,E2 -18205.293} C_VEL
LIN {X 0,Y 263.181,Z 441.328,A -85,B 0,C 180,E1 -18208.73,E2 -18208.73} C_VEL
LIN {X 0,Y 263.183,Z 441.383,A -85,B 0,C 180,E1 -18211.02,E2 -18211.02} C_VEL
LIN {X 0,Y 264.865,Z 447.384,A -85,B 0,C 180,E1 -18214.658,E2 -18214.658} C_VEL
LIN {X 0,Y 266.428,Z 453.68,A -85,B 0,C 180,E1 -18218.308,E2 -18218.308} C_VEL
LIN {X 0,Y 267.846,Z 460.3,A -85,B 0,C 180,E1 -18221.926,E2 -18221.926} C_VEL
LIN {X 0,Y 269.185,Z 467.899,A -85,B 0,C 180,E1 -18225.887,E2 -18225.887} C_VEL
LIN {X 0,Y 269.867,Z 472.905,A -85,B 0,C 180,E1 -18228.358,E2 -18228.358} C_VEL
LIN {X 0,Y 269.329,Z 478.306,A -85,B 0,C 180,E1 -18230.744,E2 -18230.744} C_VEL
LIN {X 0,Y 268.273,Z 487.848,A -85,B 0,C 180,E1 -18234.806,E2 -18234.806} C_VEL
LIN {X 0,Y 267.988,Z 491.565,A -85,B 0,C 180,E1 -18236.258,E2 -18236.258} C_VEL
LIN {X 0,Y 272.736,Z 506.767,A -85,B 0,C 180,E1 -18237.51,E2 -18237.51} C_VEL
LIN {X 0,Y 276.062,Z 520.956,A -85,B 0,C 180,E1 -18238.829,E2 -18238.829} C_VEL
LIN {X 0,Y 278.094,Z 533.582,A -85,B 0,C 180,E1 -18240.16,E2 -18240.16} C_VEL
LIN {X 0,Y 279.037,Z 544.203,A -85,B 0,C 180,E1 -18241.41,E2 -18241.41} C_VEL
LIN {X 0,Y 277.691,Z 553.74,A -85,B 0,C 180,E1 -18242.478,E2 -18242.478} C_VEL
LIN {X 0,Y 275.299,Z 565.681,A -85,B 0,C 180,E1 -18244.076,E2 -18244.076} C_VEL
LIN {X 0,Y 272.91,Z 575.528,A -85,B 0,C 180,E1 -18245.667,E2 -18245.667} C_VEL
LIN {X 0,Y 270.303,Z 586.36,A -85,B 0,C 180,E1 -18247.852,E2 -18247.852} C_VEL
LIN {X 0,Y 267.925,Z 595.301,A -85,B 0,C 180,E1 -18250.062,E2 -18250.062} C_VEL
LIN {X 0,Y 265.808,Z 603.587,A -85,B 0,C 180,E1 -18252.602,E2 -18252.602} C_VEL
LIN {X 0,Y 264.583,Z 608.943,A -85,B 0,C 180,E1 -18254.596,E2 -18254.596} C_VEL
LIN {X 0,Y 263.204,Z 614.027,A -85,B 0,C 180,E1 -18256.882,E2 -18256.882} C_VEL
LIN {X 0,Y 262.052,Z 619.354,A -85,B 0,C 180,E1 -18259.961,E2 -18259.961} C_VEL
LIN {X 0,Y 261.516,Z 622.297,A -85,B 0,C 180,E1 -18262.278,E2 -18262.278} C_VEL
LIN {X 0,Y 261.126,Z 625.012,A -85,B 0,C 180,E1 -18265.369,E2 -18265.369} C_VEL
LIN {X 0,Y 261.05,Z 626.372,A -85,B 0,C 180,E1 -18268.457,E2 -18268.457} C_VEL
LIN {X 0,Y 261.075,Z 626.554,A -85,B 0,C 180,E1 -18270,E2 -18270} C_VEL
LIN {X 0,Y 261.07,Z 625.916,A -85,B 0,C 180,E1 -18273.086,E2 -18273.086} C_VEL
LIN {X 0,Y 261.261,Z 623.932,A -85,B 0,C 180,E1 -18276.177,E2 -18276.177} C_VEL
LIN {X 0,Y 261.857,Z 620.562,A -85,B 0,C 180,E1 -18279.267,E2 -18279.267} C_VEL
LIN {X 0,Y 262.813,Z 615.707,A -85,B 0,C 180,E1 -18282.353,E2 -18282.353} C_VEL
LIN {X 0,Y 264.032,Z 610.997,A -85,B 0,C 180,E1 -18284.647,E2 -18284.647} C_VEL
LIN {X 0,Y 265.483,Z 605.271,A -85,B 0,C 180,E1 -18286.93,E2 -18286.93} C_VEL
LIN {X 0,Y 267.586,Z 597.033,A -85,B 0,C 180,E1 -18289.565,E2 -18289.565} C_VEL
LIN {X 0,Y 269.851,Z 588.437,A -85,B 0,C 180,E1 -18291.785,E2 -18291.785} C_VEL
LIN {X 0,Y 272.37,Z 578.02,A -85,B 0,C 180,E1 -18293.979,E2 -18293.979} C_VEL
LIN {X 0,Y 274.905,Z 567.512,A -85,B 0,C 180,E1 -18295.76,E2 -18295.76} C_VEL
LIN {X 0,Y 277.351,Z 555.533,A -85,B 0,C 180,E1 -18297.418,E2 -18297.418} C_VEL
LIN {X 0,Y 279.167,Z 545.211,A -85,B 0,C 180,E1 -18298.576,E2 -18298.576} C_VEL
LIN {X 0,Y 277.973,Z 532.482,A -85,B 0,C 180,E1 -18300.082,E2 -18300.082} C_VEL
LIN {X 0,Y 275.645,Z 518.581,A -85,B 0,C 180,E1 -18301.522,E2 -18301.522} C_VEL
LIN {X 0,Y 272.306,Z 505.176,A -85,B 0,C 180,E1 -18302.755,E2 -18302.755} C_VEL
LIN {X 0,Y 268.513,Z 493.424,A -85,B 0,C 180,E1 -18303.736,E2 -18303.736} C_VEL
LIN {X 0,Y 267.943,Z 491.235,A -85,B 0,C 180,E1 -18303.93,E2 -18303.93} C_VEL
LIN {X 0,Y 268.909,Z 482.293,A -85,B 0,C 180,E1 -18307.688,E2 -18307.688} C_VEL
LIN {X 0,Y 269.804,Z 474.762,A -85,B 0,C 180,E1 -18310.939,E2 -18310.939} C_VEL
LIN {X 0,Y 269.736,Z 471.128,A -85,B 0,C 180,E1 -18312.643,E2 -18312.643} C_VEL
LIN {X 0,Y 268.605,Z 464.336,A -85,B 0,C 180,E1 -18316.102,E2 -18316.102} C_VEL
LIN {X 0,Y 267.289,Z 457.642,A -85,B 0,C 180,E1 -18319.687,E2 -18319.687} C_VEL
LIN {X 0,Y 265.796,Z 450.856,A -85,B 0,C 180,E1 -18323.492,E2 -18323.492} C_VEL
LIN {X 0,Y 263.811,Z 443.565,A -85,B 0,C 180,E1 -18327.805,E2 -18327.805} C_VEL
LIN {X 0,Y 263.304,Z 442.095,A -85,B 0,C 180,E1 -18328.866,E2 -18328.866} C_VEL
LIN {X 0,Y 268.167,Z 456.577,A -85,B 0,C 180,E1 -18330.622,E2 -18330.622} C_VEL
LIN {X 0,Y 272.276,Z 470.163,A -85,B 0,C 180,E1 -18332.492,E2 -18332.492} C_VEL
LIN {X 0,Y 273.8,Z 475.563,A -85,B 0,C 180,E1 -18333.308,E2 -18333.308} C_VEL
LIN {X 0,Y 273.505,Z 479.894,A -85,B 0,C 180,E1 -18333.893,E2 -18333.893} C_VEL
LIN {X 0,Y 271.388,Z 493.73,A -85,B 0,C 180,E1 -18335.929,E2 -18335.929} C_VEL
LIN {X 0,Y 269.321,Z 506.329,A -85,B 0,C 180,E1 -18338.17,E2 -18338.17} C_VEL
LIN {X 0,Y 267.509,Z 516.897,A -85,B 0,C 180,E1 -18340.429,E2 -18340.429} C_VEL
LIN {X 0,Y 266.042,Z 526.048,A -85,B 0,C 180,E1 -18342.748,E2 -18342.748} C_VEL
LIN {X 0,Y 264.891,Z 533.661,A -85,B 0,C 180,E1 -18345.008,E2 -18345.008} C_VEL
LIN {X 0,Y 263.818,Z 541.302,A -85,B 0,C 180,E1 -18347.695,E2 -18347.695} C_VEL
LIN {X 0,Y 263.004,Z 548.42,A -85,B 0,C 180,E1 -18350.774,E2 -18350.774} C_VEL
LIN {X 0,Y 262.512,Z 554.032,A -85,B 0,C 180,E1 -18353.852,E2 -18353.852} C_VEL
LIN {X 0,Y 262.353,Z 557.506,A -85,B 0,C 180,E1 -18356.342,E2 -18356.342} C_VEL
LIN {X 0,Y 261.591,Z 559.054,A -85,B 0,C 180,E1 -18357.577,E2 -18357.577} C_VEL
LIN {X 0,Y 258.682,Z 561.254,A -85,B 0,C 180,E1 -18359.607,E2 -18359.607} C_VEL
LIN {X 0,Y 256.368,Z 562.692,A -85,B 0,C 180,E1 -18361.273,E2 -18361.273} C_VEL
LIN {X 0,Y 255.52,Z 563.5,A -85,B 0,C 180,E1 -18362.573,E2 -18362.573} C_VEL
LIN {X 0,Y 255.525,Z 563.735,A -85,B 0,C 180,E1 -18363.012,E2 -18363.012} C_VEL
LIN {X 0,Y 256.518,Z 564.558,A -85,B 0,C 180,E1 -18366.292,E2 -18366.292} C_VEL
LIN {X 0,Y 257.864,Z 564.157,A -85,B 0,C 180,E1 -18369.412,E2 -18369.412} C_VEL
LIN {X 0,Y 259.574,Z 562.653,A -85,B 0,C 180,E1 -18372.509,E2 -18372.509} C_VEL
LIN {X 0,Y 261.792,Z 560.03,A -85,B 0,C 180,E1 -18375.572,E2 -18375.572} C_VEL
LIN {X 0,Y 264.73,Z 556.183,A -85,B 0,C 180,E1 -18378.577,E2 -18378.577} C_VEL
LIN {X 0,Y 268.189,Z 551.157,A -85,B 0,C 180,E1 -18381.523,E2 -18381.523} C_VEL
LIN {X 0,Y 272.507,Z 544.714,A -85,B 0,C 180,E1 -18384.371,E2 -18384.371} C_VEL
LIN {X 0,Y 277.305,Z 536.871,A -85,B 0,C 180,E1 -18387.141,E2 -18387.141} C_VEL
LIN {X 0,Y 281.943,Z 528.828,A -85,B 0,C 180,E1 -18389.451,E2 -18389.451} C_VEL
LIN {X 0,Y 287.314,Z 519.085,A -85,B 0,C 180,E1 -18391.73,E2 -18391.73} C_VEL
LIN {X 0,Y 293.696,Z 506.467,A -85,B 0,C 180,E1 -18394.099,E2 -18394.099} C_VEL
LIN {X 0,Y 293.875,Z 502.643,A -85,B 0,C 180,E1 -18395.599,E2 -18395.599} C_VEL
LIN {X 0,Y 293.75,Z 500.308,A -85,B 0,C 180,E1 -18396.736,E2 -18396.736} C_VEL
LIN {X 0,Y 293.207,Z 499.153,A -85,B 0,C 180,E1 -18397.722,E2 -18397.722} C_VEL
LIN {X 0,Y 291.964,Z 498.071,A -85,B 0,C 180,E1 -18399.62,E2 -18399.62} C_VEL
LIN {X 0,Y 290.768,Z 498.171,A -85,B 0,C 180,E1 -18401.472,E2 -18401.472} C_VEL
LIN {X 0,Y 289.59,Z 499.585,A -85,B 0,C 180,E1 -18403.276,E2 -18403.276} C_VEL
LIN {X 0,Y 288.951,Z 500.848,A -85,B 0,C 180,E1 -18404.161,E2 -18404.161} C_VEL
LIN {X 0,Y 286.907,Z 507.314,A -85,B 0,C 180,E1 -18407.296,E2 -18407.296} C_VEL
LIN {X 0,Y 285.751,Z 513.709,A -85,B 0,C 180,E1 -18409.68,E2 -18409.68} C_VEL
LIN {X 0,Y 284.564,Z 521.105,A -85,B 0,C 180,E1 -18411.871,E2 -18411.871} C_VEL
LIN {X 0,Y 283.139,Z 529.12,A -85,B 0,C 180,E1 -18413.909,E2 -18413.909} C_VEL
LIN {X 0,Y 280.929,Z 538.338,A -85,B 0,C 180,E1 -18415.963,E2 -18415.963} C_VEL
LIN {X 0,Y 277.253,Z 549.447,A -85,B 0,C 180,E1 -18418.265,E2 -18418.265} C_VEL
LIN {X 0,Y 274.137,Z 558.988,A -85,B 0,C 180,E1 -18420.429,E2 -18420.429} C_VEL
LIN {X 0,Y 273.409,Z 561.048,A -85,B 0,C 180,E1 -18420.924,E2 -18420.924} C_VEL
LIN {X 0,Y 268.855,Z 570.72,A -85,B 0,C 180,E1 -18423.197,E2 -18423.197} C_VEL
LIN {X 0,Y 267.21,Z 574.523,A -85,B 0,C 180,E1 -18424.175,E2 -18424.175} C_VEL
LIN {X 0,Y 264.535,Z 585.073,A -85,B 0,C 180,E1 -18426.099,E2 -18426.099} C_VEL
LIN {X 0,Y 262.006,Z 595.019,A -85,B 0,C 180,E1 -18428.357,E2 -18428.357} C_VEL
LIN {X 0,Y 259.75,Z 603.259,A -85,B 0,C 180,E1 -18430.643,E2 -18430.643} C_VEL
LIN {X 0,Y 257.796,Z 611.124,A -85,B 0,C 180,E1 -18433.366,E2 -18433.366} C_VEL
LIN {X 0,Y 256.401,Z 616.626,A -85,B 0,C 180,E1 -18435.718,E2 -18435.718} C_VEL
LIN {X 0,Y 255.061,Z 622.38,A -85,B 0,C 180,E1 -18438.879,E2 -18438.879} C_VEL
LIN {X 0,Y 254.344,Z 626.555,A -85,B 0,C 180,E1 -18442.059,E2 -18442.059} C_VEL
LIN {X 0,Y 254.013,Z 629.282,A -85,B 0,C 180,E1 -18445.239,E2 -18445.239} C_VEL
LIN {X 0,Y 254.022,Z 630.636,A -85,B 0,C 180,E1 -18448.415,E2 -18448.415} C_VEL
LIN {X 0,Y 254.048,Z 630.803,A -85,B 0,C 180,E1 -18450,E2 -18450} C_VEL
LIN {X 0,Y 253.992,Z 630.118,A -85,B 0,C 180,E1 -18453.172,E2 -18453.172} C_VEL
LIN {X 0,Y 254.154,Z 628.077,A -85,B 0,C 180,E1 -18456.35,E2 -18456.35} C_VEL
LIN {X 0,Y 254.635,Z 624.627,A -85,B 0,C 180,E1 -18459.532,E2 -18459.532} C_VEL
LIN {X 0,Y 255.575,Z 619.665,A -85,B 0,C 180,E1 -18462.708,E2 -18462.708} C_VEL
LIN {X 0,Y 256.829,Z 614.854,A -85,B 0,C 180,E1 -18465.068,E2 -18465.068} C_VEL
LIN {X 0,Y 258.571,Z 607.485,A -85,B 0,C 180,E1 -18467.954,E2 -18467.954} C_VEL
LIN {X 0,Y 260.795,Z 599.244,A -85,B 0,C 180,E1 -18470.507,E2 -18470.507} C_VEL
LIN {X 0,Y 263.155,Z 590.181,A -85,B 0,C 180,E1 -18472.783,E2 -18472.783} C_VEL
LIN {X 0,Y 265.973,Z 579.171,A -85,B 0,C 180,E1 -18475.01,E2 -18475.01} C_VEL
LIN {X 0,Y 268.468,Z 568.758,A -85,B 0,C 180,E1 -18476.703,E2 -18476.703} C_VEL
LIN {X 0,Y 270.733,Z 556.985,A -85,B 0,C 180,E1 -18478.278,E2 -18478.278} C_VEL
LIN {X 0,Y 270.479,Z 544.704,A -85,B 0,C 180,E1 -18479.858,E2 -18479.858} C_VEL
LIN {X 0,Y 269.431,Z 531.388,A -85,B 0,C 180,E1 -18481.321,E2 -18481.321} C_VEL
LIN {X 0,Y 267.755,Z 516.934,A -85,B 0,C 180,E1 -18482.619,E2 -18482.619} C_VEL
LIN {X 0,Y 264.264,Z 503.439,A -85,B 0,C 180,E1 -18483.787,E2 -18483.787} C_VEL
LIN {X 0,Y 259.766,Z 490.222,A -85,B 0,C 180,E1 -18484.915,E2 -18484.915} C_VEL
LIN {X 0,Y 258.691,Z 480.302,A -85,B 0,C 180,E1 -18487.238,E2 -18487.238} C_VEL
LIN {X 0,Y 257.366,Z 470.197,A -85,B 0,C 180,E1 -18489.719,E2 -18489.719} C_VEL
LIN {X 0,Y 258.149,Z 464.324,A -85,B 0,C 180,E1 -18493.956,E2 -18493.956} C_VEL
LIN {X 0,Y 258.738,Z 459.871,A -85,B 0,C 180,E1 -18497.229,E2 -18497.229} C_VEL
LIN {X 0,Y 258.57,Z 455.692,A -85,B 0,C 180,E1 -18500.415,E2 -18500.415} C_VEL
LIN {X 0,Y 257.508,Z 449.975,A -85,B 0,C 180,E1 -18505.031,E2 -18505.031} C_VEL
LIN {X 0,Y 256.631,Z 444.626,A -85,B 0,C 180,E1 -18509.56,E2 -18509.56} C_VEL
LIN {X 0,Y 256.224,Z 442.194,A -85,B 0,C 180,E1 -18511.766,E2 -18511.766} C_VEL
LIN {X 0,Y 256.169,Z 442.194,A -85,B 0,C 180,E1 -18515.699,E2 -18515.699} C_VEL
LIN {X 0,Y 256.168,Z 442.178,A -85,B 0,C 180,E1 -18519.105,E2 -18519.105} C_VEL
LIN {X 0,Y 256.301,Z 442.166,A -85,B 0,C 180,E1 -18524.085,E2 -18524.085} C_VEL
LIN {X 0,Y 256.297,Z 442.18,A -85,B 0,C 180,E1 -18528.934,E2 -18528.934} C_VEL
LIN {X 0,Y 256.503,Z 442.139,A -85,B 0,C 180,E1 -18532.126,E2 -18532.126} C_VEL
LIN {X 0,Y 256.499,Z 442.135,A -85,B 0,C 180,E1 -18536.859,E2 -18536.859} C_VEL
LIN {X 0,Y 256.775,Z 442.127,A -85,B 0,C 180,E1 -18540,E2 -18540} C_VEL
LIN {X 0,Y 256.499,Z 442.136,A -85,B 0,C 180,E1 -18543.141,E2 -18543.141} C_VEL
LIN {X 0,Y 256.542,Z 442.135,A -85,B 0,C 180,E1 -18547.873,E2 -18547.873} C_VEL
LIN {X 0,Y 256.312,Z 442.185,A -85,B 0,C 180,E1 -18551.066,E2 -18551.066} C_VEL
LIN {X 0,Y 256.302,Z 442.185,A -85,B 0,C 180,E1 -18555.915,E2 -18555.915} C_VEL
LIN {X 0,Y 256.164,Z 442.205,A -85,B 0,C 180,E1 -18560.896,E2 -18560.896} C_VEL
LIN {X 0,Y 256.172,Z 442.201,A -85,B 0,C 180,E1 -18565.13,E2 -18565.13} C_VEL
LIN {X 0,Y 256.11,Z 442.242,A -85,B 0,C 180,E1 -18569.456,E2 -18569.456} C_VEL
LIN {X 0,Y 257.66,Z 447.817,A -85,B 0,C 180,E1 -18573.061,E2 -18573.061} C_VEL
LIN {X 0,Y 258.731,Z 451.704,A -85,B 0,C 180,E1 -18575.422,E2 -18575.422} C_VEL
LIN {X 0,Y 259.947,Z 456.771,A -85,B 0,C 180,E1 -18578.45,E2 -18578.45} C_VEL
LIN {X 0,Y 261.609,Z 464.794,A -85,B 0,C 180,E1 -18582.887,E2 -18582.887} C_VEL
LIN {X 0,Y 262.968,Z 473.009,A -85,B 0,C 180,E1 -18587.166,E2 -18587.166} C_VEL
LIN {X 0,Y 263.131,Z 475.565,A -85,B 0,C 180,E1 -18588.405,E2 -18588.405} C_VEL
LIN {X 0,Y 262.197,Z 483.524,A -85,B 0,C 180,E1 -18591.939,E2 -18591.939} C_VEL
LIN {X 0,Y 261.351,Z 491.462,A -85,B 0,C 180,E1 -18595.279,E2 -18595.279} C_VEL
LIN {X 0,Y 266.071,Z 506.281,A -85,B 0,C 180,E1 -18596.565,E2 -18596.565} C_VEL
LIN {X 0,Y 269.257,Z 519.464,A -85,B 0,C 180,E1 -18597.833,E2 -18597.833} C_VEL
LIN {X 0,Y 271.471,Z 532.702,A -85,B 0,C 180,E1 -18599.264,E2 -18599.264} C_VEL
LIN {X 0,Y 272.55,Z 544.247,A -85,B 0,C 180,E1 -18600.664,E2 -18600.664} C_VEL
LIN {X 0,Y 272.312,Z 548.634,A -85,B 0,C 180,E1 -18601.184,E2 -18601.184} C_VEL
LIN {X 0,Y 269.993,Z 560.741,A -85,B 0,C 180,E1 -18602.691,E2 -18602.691} C_VEL
LIN {X 0,Y 267.25,Z 572.442,A -85,B 0,C 180,E1 -18604.493,E2 -18604.493} C_VEL
LIN {X 0,Y 264.568,Z 583.022,A -85,B 0,C 180,E1 -18606.518,E2 -18606.518} C_VEL
LIN {X 0,Y 262.032,Z 592.558,A -85,B 0,C 180,E1 -18608.772,E2 -18608.772} C_VEL
LIN {X 0,Y 259.792,Z 600.464,A -85,B 0,C 180,E1 -18611.057,E2 -18611.057} C_VEL
LIN {X 0,Y 258.295,Z 607.037,A -85,B 0,C 180,E1 -18613.399,E2 -18613.399} C_VEL
LIN {X 0,Y 256.678,Z 612.494,A -85,B 0,C 180,E1 -18615.734,E2 -18615.734} C_VEL
LIN {X 0,Y 255.3,Z 618.204,A -85,B 0,C 180,E1 -18618.89,E2 -18618.89} C_VEL
LIN {X 0,Y 254.452,Z 622.356,A -85,B 0,C 180,E1 -18622.062,E2 -18622.062} C_VEL
LIN {X 0,Y 254.063,Z 625.071,A -85,B 0,C 180,E1 -18625.24,E2 -18625.24} C_VEL
LIN {X 0,Y 253.961,Z 626.431,A -85,B 0,C 180,E1 -18628.414,E2 -18628.414} C_VEL
LIN {X 0,Y 253.982,Z 626.612,A -85,B 0,C 180,E1 -18630,E2 -18630} C_VEL
LIN {X 0,Y 253.971,Z 625.974,A -85,B 0,C 180,E1 -18633.173,E2 -18633.173} C_VEL
LIN {X 0,Y 254.183,Z 623.99,A -85,B 0,C 180,E1 -18636.35,E2 -18636.35} C_VEL
LIN {X 0,Y 254.82,Z 620.619,A -85,B 0,C 180,E1 -18639.525,E2 -18639.525} C_VEL
LIN {X 0,Y 255.833,Z 615.763,A -85,B 0,C 180,E1 -18642.695,E2 -18642.695} C_VEL
LIN {X 0,Y 257.146,Z 611.053,A -85,B 0,C 180,E1 -18645.049,E2 -18645.049} C_VEL
LIN {X 0,Y 258.994,Z 604.082,A -85,B 0,C 180,E1 -18647.828,E2 -18647.828} C_VEL
LIN {X 0,Y 261.205,Z 595.75,A -85,B 0,C 180,E1 -18650.474,E2 -18650.474} C_VEL
LIN {X 0,Y 263.618,Z 586.884,A -85,B 0,C 180,E1 -18652.741,E2 -18652.741} C_VEL
LIN {X 0,Y 266.376,Z 576.149,A -85,B 0,C 180,E1 -18654.97,E2 -18654.97} C_VEL
LIN {X 0,Y 269.096,Z 565.248,A -85,B 0,C 180,E1 -18656.777,E2 -18656.777} C_VEL
LIN {X 0,Y 271.384,Z 554.081,A -85,B 0,C 180,E1 -18658.297,E2 -18658.297} C_VEL
LIN {X 0,Y 272.689,Z 547.102,A -85,B 0,C 180,E1 -18659.091,E2 -18659.091} C_VEL
LIN {X 0,Y 271.984,Z 536.515,A -85,B 0,C 180,E1 -18660.413,E2 -18660.413} C_VEL
LIN {X 0,Y 270.259,Z 524.547,A -85,B 0,C 180,E1 -18661.763,E2 -18661.763} C_VEL
LIN {X 0,Y 267.531,Z 511.727,A -85,B 0,C 180,E1 -18663.055,E2 -18663.055} C_VEL
LIN {X 0,Y 263.978,Z 499.336,A -85,B 0,C 180,E1 -18664.181,E2 -18664.181} C_VEL
LIN {X 0,Y 261.355,Z 491.241,A -85,B 0,C 180,E1 -18664.9,E2 -18664.9} C_VEL
LIN {X 0,Y 262.433,Z 481.59,A -85,B 0,C 180,E1 -18669.047,E2 -18669.047} C_VEL
LIN {X 0,Y 263.122,Z 475.885,A -85,B 0,C 180,E1 -18671.593,E2 -18671.593} C_VEL
LIN {X 0,Y 262.768,Z 471.469,A -85,B 0,C 180,E1 -18673.768,E2 -18673.768} C_VEL
LIN {X 0,Y 261.442,Z 463.889,A -85,B 0,C 180,E1 -18677.775,E2 -18677.775} C_VEL
LIN {X 0,Y 260.04,Z 457.008,A -85,B 0,C 180,E1 -18681.607,E2 -18681.607} C_VEL
LIN {X 0,Y 258.861,Z 452.081,A -85,B 0,C 180,E1 -18684.537,E2 -18684.537} C_VEL
LIN {X 0,Y 257.032,Z 445.462,A -85,B 0,C 180,E1 -18688.658,E2 -18688.658} C_VEL
LIN {X 0,Y 261.815,Z 459.741,A -85,B 0,C 180,E1 -18690.502,E2 -18690.502} C_VEL
LIN {X 0,Y 265.613,Z 472.426,A -85,B 0,C 180,E1 -18692.325,E2 -18692.325} C_VEL
LIN {X 0,Y 266.985,Z 478.071,A -85,B 0,C 180,E1 -18693.188,E2 -18693.188} C_VEL
LIN {X 0,Y 264.963,Z 491.191,A -85,B 0,C 180,E1 -18695.097,E2 -18695.097} C_VEL
LIN {X 0,Y 262.925,Z 503.26,A -85,B 0,C 180,E1 -18697.195,E2 -18697.195} C_VEL
LIN {X 0,Y 261.057,Z 514.436,A -85,B 0,C 180,E1 -18699.514,E2 -18699.514} C_VEL
LIN {X 0,Y 259.29,Z 524.596,A -85,B 0,C 180,E1 -18702.02,E2 -18702.02} C_VEL
LIN {X 0,Y 258.002,Z 533.364,A -85,B 0,C 180,E1 -18704.598,E2 -18704.598} C_VEL
LIN {X 0,Y 256.844,Z 541.222,A -85,B 0,C 180,E1 -18707.355,E2 -18707.355} C_VEL
LIN {X 0,Y 255.957,Z 548.51,A -85,B 0,C 180,E1 -18710.517,E2 -18710.517} C_VEL
LIN {X 0,Y 255.463,Z 554.281,A -85,B 0,C 180,E1 -18713.682,E2 -18713.682} C_VEL
LIN {X 0,Y 255.302,Z 557.985,A -85,B 0,C 180,E1 -18716.278,E2 -18716.278} C_VEL
LIN {X 0,Y 255.149,Z 560.429,A -85,B 0,C 180,E1 -18718.421,E2 -18718.421} C_VEL
LIN {X 0,Y 255.301,Z 562.981,A -85,B 0,C 180,E1 -18721.577,E2 -18721.577} C_VEL
LIN {X 0,Y 255.525,Z 563.735,A -85,B 0,C 180,E1 -18723.012,E2 -18723.012} C_VEL
LIN {X 0,Y 255.191,Z 564.39,A -85,B 0,C 180,E1 -18724.327,E2 -18724.327} C_VEL
LIN {X 0,Y 253.066,Z 565.187,A -85,B 0,C 180,E1 -18726.504,E2 -18726.504} C_VEL
LIN {X 0,Y 251.397,Z 565.414,A -85,B 0,C 180,E1 -18728.273,E2 -18728.273} C_VEL
LIN {X 0,Y 251.009,Z 565.261,A -85,B 0,C 180,E1 -18729.623,E2 -18729.623} C_VEL
LIN {X 0,Y 251.156,Z 565.132,A -85,B 0,C 180,E1 -18730.072,E2 -18730.072} C_VEL
LIN {X 0,Y 252.786,Z 563.97,A -85,B 0,C 180,E1 -18732.851,E2 -18732.851} C_VEL
LIN {X 0,Y 255.129,Z 561.573,A -85,B 0,C 180,E1 -18735.99,E2 -18735.99} C_VEL
LIN {X 0,Y 258.234,Z 558.006,A -85,B 0,C 180,E1 -18739.062,E2 -18739.062} C_VEL
LIN {X 0,Y 261.891,Z 553.234,A -85,B 0,C 180,E1 -18742.067,E2 -18742.067} C_VEL
LIN {X 0,Y 266.425,Z 547.119,A -85,B 0,C 180,E1 -18744.965,E2 -18744.965} C_VEL
LIN {X 0,Y 271.492,Z 539.672,A -85,B 0,C 180,E1 -18747.772,E2 -18747.772} C_VEL
LIN {X 0,Y 277.169,Z 530.709,A -85,B 0,C 180,E1 -18750.473,E2 -18750.473} C_VEL
LIN {X 0,Y 283.61,Z 519.953,A -85,B 0,C 180,E1 -18753.036,E2 -18753.036} C_VEL
LIN {X 0,Y 288.269,Z 511.526,A -85,B 0,C 180,E1 -18754.669,E2 -18754.669} C_VEL
LIN {X 0,Y 289.122,Z 509.647,A -85,B 0,C 180,E1 -18755.115,E2 -18755.115} C_VEL
LIN {X 0,Y 289.346,Z 506.243,A -85,B 0,C 180,E1 -18756.722,E2 -18756.722} C_VEL
LIN {X 0,Y 289.154,Z 505.271,A -85,B 0,C 180,E1 -18757.419,E2 -18757.419} C_VEL
LIN {X 0,Y 288.101,Z 504.012,A -85,B 0,C 180,E1 -18759.364,E2 -18759.364} C_VEL
LIN {X 0,Y 286.801,Z 504.156,A -85,B 0,C 180,E1 -18761.424,E2 -18761.424} C_VEL
LIN {X 0,Y 286.095,Z 504.946,A -85,B 0,C 180,E1 -18762.527,E2 -18762.527} C_VEL
LIN {X 0,Y 285.224,Z 506.292,A -85,B 0,C 180,E1 -18763.624,E2 -18763.624} C_VEL
LIN {X 0,Y 282.625,Z 513.172,A -85,B 0,C 180,E1 -18767.091,E2 -18767.091} C_VEL
LIN {X 0,Y 281.025,Z 519.539,A -85,B 0,C 180,E1 -18769.442,E2 -18769.442} C_VEL
LIN {X 0,Y 279.505,Z 526.443,A -85,B 0,C 180,E1 -18771.559,E2 -18771.559} C_VEL
LIN {X 0,Y 277.261,Z 535.42,A -85,B 0,C 180,E1 -18773.89,E2 -18773.89} C_VEL
LIN {X 0,Y 274.691,Z 543.52,A -85,B 0,C 180,E1 -18775.745,E2 -18775.745} C_VEL
LIN {X 0,Y 269.172,Z 557.714,A -85,B 0,C 180,E1 -18778.958,E2 -18778.958} C_VEL
LIN {X 0,Y 267.656,Z 562.064,A -85,B 0,C 180,E1 -18780.073,E2 -18780.073} C_VEL
LIN {X 0,Y 262.616,Z 571.833,A -85,B 0,C 180,E1 -18782.507,E2 -18782.507} C_VEL
LIN {X 0,Y 260.257,Z 576.618,A -85,B 0,C 180,E1 -18783.864,E2 -18783.864} C_VEL
LIN {X 0,Y 257.53,Z 586.798,A -85,B 0,C 180,E1 -18785.836,E2 -18785.836} C_VEL
LIN {X 0,Y 254.983,Z 596.448,A -85,B 0,C 180,E1 -18788.155,E2 -18788.155} C_VEL
LIN {X 0,Y 252.706,Z 604.434,A -85,B 0,C 180,E1 -18790.505,E2 -18790.505} C_VEL
LIN {X 0,Y 250.981,Z 611.07,A -85,B 0,C 180,E1 -18792.901,E2 -18792.901} C_VEL
LIN {X 0,Y 249.487,Z 616.57,A -85,B 0,C 180,E1 -18795.314,E2 -18795.314} C_VEL
LIN {X 0,Y 248.068,Z 622.323,A -85,B 0,C 180,E1 -18798.561,E2 -18798.561} C_VEL
LIN {X 0,Y 247.285,Z 626.498,A -85,B 0,C 180,E1 -18801.83,E2 -18801.83} C_VEL
LIN {X 0,Y 246.922,Z 629.224,A -85,B 0,C 180,E1 -18805.102,E2 -18805.102} C_VEL
LIN {X 0,Y 246.93,Z 630.577,A -85,B 0,C 180,E1 -18808.369,E2 -18808.369} C_VEL
LIN {X 0,Y 246.956,Z 630.744,A -85,B 0,C 180,E1 -18810,E2 -18810} C_VEL
LIN {X 0,Y 246.894,Z 630.06,A -85,B 0,C 180,E1 -18813.264,E2 -18813.264} C_VEL
LIN {X 0,Y 247.066,Z 628.017,A -85,B 0,C 180,E1 -18816.533,E2 -18816.533} C_VEL
LIN {X 0,Y 247.602,Z 624.568,A -85,B 0,C 180,E1 -18819.806,E2 -18819.806} C_VEL
LIN {X 0,Y 248.609,Z 619.606,A -85,B 0,C 180,E1 -18823.071,E2 -18823.071} C_VEL
LIN {X 0,Y 249.938,Z 614.795,A -85,B 0,C 180,E1 -18825.494,E2 -18825.494} C_VEL
LIN {X 0,Y 251.679,Z 607.861,A -85,B 0,C 180,E1 -18828.299,E2 -18828.299} C_VEL
LIN {X 0,Y 254.118,Z 599.187,A -85,B 0,C 180,E1 -18831.072,E2 -18831.072} C_VEL
LIN {X 0,Y 256.606,Z 590.126,A -85,B 0,C 180,E1 -18833.399,E2 -18833.399} C_VEL
LIN {X 0,Y 258.995,Z 581.08,A -85,B 0,C 180,E1 -18835.302,E2 -18835.302} C_VEL
LIN {X 0,Y 261.715,Z 570.268,A -85,B 0,C 180,E1 -18837.162,E2 -18837.162} C_VEL
LIN {X 0,Y 264.202,Z 558.414,A -85,B 0,C 180,E1 -18838.825,E2 -18838.825} C_VEL
LIN {X 0,Y 264.168,Z 547.021,A -85,B 0,C 180,E1 -18840.363,E2 -18840.363} C_VEL
LIN {X 0,Y 263.329,Z 533.7,A -85,B 0,C 180,E1 -18841.921,E2 -18841.921} C_VEL
LIN {X 0,Y 261.896,Z 519.621,A -85,B 0,C 180,E1 -18843.27,E2 -18843.27} C_VEL
LIN {X 0,Y 258.722,Z 506.494,A -85,B 0,C 180,E1 -18844.489,E2 -18844.489} C_VEL
LIN {X 0,Y 253.245,Z 490.051,A -85,B 0,C 180,E1 -18846.002,E2 -18846.002} C_VEL
LIN {X 0,Y 251.801,Z 477.498,A -85,B 0,C 180,E1 -18849.139,E2 -18849.139} C_VEL
LIN {X 0,Y 251.018,Z 472.206,A -85,B 0,C 180,E1 -18850.504,E2 -18850.504} C_VEL
LIN {X 0,Y 250.621,Z 467.999,A -85,B 0,C 180,E1 -18851.651,E2 -18851.651} C_VEL
LIN {X 0,Y 251.404,Z 462.595,A -85,B 0,C 180,E1 -18855.663,E2 -18855.663} C_VEL
LIN {X 0,Y 251.7,Z 459.632,A -85,B 0,C 180,E1 -18857.923,E2 -18857.923} C_VEL
LIN {X 0,Y 251.559,Z 456.977,A -85,B 0,C 180,E1 -18860.016,E2 -18860.016} C_VEL
LIN {X 0,Y 250.623,Z 451.598,A -85,B 0,C 180,E1 -18864.412,E2 -18864.412} C_VEL
LIN {X 0,Y 249.755,Z 446.677,A -85,B 0,C 180,E1 -18868.629,E2 -18868.629} C_VEL
LIN {X 0,Y 249.181,Z 443.068,A -85,B 0,C 180,E1 -18871.923,E2 -18871.923} C_VEL
LIN {X 0,Y 249.153,Z 443.057,A -85,B 0,C 180,E1 -18874.969,E2 -18874.969} C_VEL
LIN {X 0,Y 249.112,Z 443.059,A -85,B 0,C 180,E1 -18880.212,E2 -18880.212} C_VEL
LIN {X 0,Y 249.243,Z 443.05,A -85,B 0,C 180,E1 -18883.622,E2 -18883.622} C_VEL
LIN {X 0,Y 249.245,Z 443.062,A -85,B 0,C 180,E1 -18888.616,E2 -18888.616} C_VEL
LIN {X 0,Y 249.445,Z 443.016,A -85,B 0,C 180,E1 -18891.902,E2 -18891.902} C_VEL
LIN {X 0,Y 249.296,Z 443.049,A -85,B 0,C 180,E1 -18895.149,E2 -18895.149} C_VEL
LIN {X 0,Y 249.677,Z 442.992,A -85,B 0,C 180,E1 -18898.387,E2 -18898.387} C_VEL
LIN {X 0,Y 249.677,Z 442.994,A -85,B 0,C 180,E1 -18901.613,E2 -18901.613} C_VEL
LIN {X 0,Y 249.452,Z 443.03,A -85,B 0,C 180,E1 -18906.755,E2 -18906.755} C_VEL
LIN {X 0,Y 249.39,Z 443.029,A -85,B 0,C 180,E1 -18909.735,E2 -18909.735} C_VEL
LIN {X 0,Y 249.207,Z 443.053,A -85,B 0,C 180,E1 -18914.703,E2 -18914.703} C_VEL
LIN {X 0,Y 249.14,Z 443.062,A -85,B 0,C 180,E1 -18918.077,E2 -18918.077} C_VEL
LIN {X 0,Y 249.086,Z 443.079,A -85,B 0,C 180,E1 -18921.518,E2 -18921.518} C_VEL
LIN {X 0,Y 249.119,Z 443.075,A -85,B 0,C 180,E1 -18925.476,E2 -18925.476} C_VEL
LIN {X 0,Y 249.093,Z 443.076,A -85,B 0,C 180,E1 -18927.745,E2 -18927.745} C_VEL
LIN {X 0,Y 250.986,Z 449.57,A -85,B 0,C 180,E1 -18932.143,E2 -18932.143} C_VEL
LIN {X 0,Y 252.618,Z 456.059,A -85,B 0,C 180,E1 -18936.216,E2 -18936.216} C_VEL
LIN {X 0,Y 253.854,Z 461.667,A -85,B 0,C 180,E1 -18939.551,E2 -18939.551} C_VEL
LIN {X 0,Y 254.92,Z 466.836,A -85,B 0,C 180,E1 -18942.488,E2 -18942.488} C_VEL
LIN {X 0,Y 256.188,Z 474.656,A -85,B 0,C 180,E1 -18946.699,E2 -18946.699} C_VEL
LIN {X 0,Y 256.448,Z 477.304,A -85,B 0,C 180,E1 -18948.026,E2 -18948.026} C_VEL
LIN {X 0,Y 255.448,Z 485.606,A -85,B 0,C 180,E1 -18951.755,E2 -18951.755} C_VEL
LIN {X 0,Y 254.82,Z 491.545,A -85,B 0,C 180,E1 -18954.259,E2 -18954.259} C_VEL
LIN {X 0,Y 259.793,Z 506.959,A -85,B 0,C 180,E1 -18955.683,E2 -18955.683} C_VEL
LIN {X 0,Y 263.042,Z 520.729,A -85,B 0,C 180,E1 -18957.075,E2 -18957.075} C_VEL
LIN {X 0,Y 265.179,Z 533.873,A -85,B 0,C 180,E1 -18958.568,E2 -18958.568} C_VEL
LIN {X 0,Y 266.198,Z 545.883,A -85,B 0,C 180,E1 -18960.094,E2 -18960.094} C_VEL
LIN {X 0,Y 266.046,Z 548.965,A -85,B 0,C 180,E1 -18960.479,E2 -18960.479} C_VEL
LIN {X 0,Y 263.702,Z 560.79,A -85,B 0,C 180,E1 -18961.983,E2 -18961.983} C_VEL
LIN {X 0,Y 260.852,Z 572.495,A -85,B 0,C 180,E1 -18963.821,E2 -18963.821} C_VEL
LIN {X 0,Y 258.047,Z 583.076,A -85,B 0,C 180,E1 -18965.887,E2 -18965.887} C_VEL
LIN {X 0,Y 255.395,Z 592.614,A -85,B 0,C 180,E1 -18968.192,E2 -18968.192} C_VEL
LIN {X 0,Y 253.065,Z 600.521,A -85,B 0,C 180,E1 -18970.533,E2 -18970.533} C_VEL
LIN {X 0,Y 251.45,Z 607.095,A -85,B 0,C 180,E1 -18972.934,E2 -18972.934} C_VEL
LIN {X 0,Y 249.793,Z 612.552,A -85,B 0,C 180,E1 -18975.332,E2 -18975.332} C_VEL
LIN {X 0,Y 248.297,Z 618.263,A -85,B 0,C 180,E1 -18978.572,E2 -18978.572} C_VEL
LIN {X 0,Y 247.401,Z 622.415,A -85,B 0,C 180,E1 -18981.834,E2 -18981.834} C_VEL
LIN {X 0,Y 246.971,Z 625.13,A -85,B 0,C 180,E1 -18985.103,E2 -18985.103} C_VEL
LIN {X 0,Y 246.874,Z 626.49,A -85,B 0,C 180,E1 -18988.369,E2 -18988.369} C_VEL
LIN {X 0,Y 246.893,Z 626.671,A -85,B 0,C 180,E1 -18990,E2 -18990} C_VEL
LIN {X 0,Y 246.875,Z 626.032,A -85,B 0,C 180,E1 -18993.264,E2 -18993.264} C_VEL
LIN {X 0,Y 247.121,Z 624.047,A -85,B 0,C 180,E1 -18996.532,E2 -18996.532} C_VEL
LIN {X 0,Y 247.806,Z 620.676,A -85,B 0,C 180,E1 -18999.797,E2 -18999.797} C_VEL
LIN {X 0,Y 248.869,Z 615.82,A -85,B 0,C 180,E1 -19003.057,E2 -19003.057} C_VEL
LIN {X 0,Y 250.848,Z 609.321,A -85,B 0,C 180,E1 -19006.27,E2 -19006.27} C_VEL
LIN {X 0,Y 252.725,Z 602.26,A -85,B 0,C 180,E1 -19009.002,E2 -19009.002} C_VEL
LIN {X 0,Y 254.929,Z 594.467,A -85,B 0,C 180,E1 -19011.425,E2 -19011.425} C_VEL
LIN {X 0,Y 257.496,Z 585.325,A -85,B 0,C 180,E1 -19013.74,E2 -19013.74} C_VEL
LIN {X 0,Y 260.234,Z 575.203,A -85,B 0,C 180,E1 -19015.816,E2 -19015.816} C_VEL
LIN {X 0,Y 263.02,Z 564.048,A -85,B 0,C 180,E1 -19017.663,E2 -19017.663} C_VEL
LIN {X 0,Y 265.593,Z 551.744,A -85,B 0,C 180,E1 -19019.309,E2 -19019.309} C_VEL
LIN {X 0,Y 266.355,Z 546.996,A -85,B 0,C 180,E1 -19019.87,E2 -19019.87} C_VEL
LIN {X 0,Y 265.254,Z 534.146,A -85,B 0,C 180,E1 -19021.522,E2 -19021.522} C_VEL
LIN {X 0,Y 263.067,Z 520.514,A -85,B 0,C 180,E1 -19023.068,E2 -19023.068} C_VEL
LIN {X 0,Y 259.658,Z 506.375,A -85,B 0,C 180,E1 -19024.5,E2 -19024.5} C_VEL
LIN {X 0,Y 254.786,Z 491.343,A -85,B 0,C 180,E1 -19025.887,E2 -19025.887} C_VEL
LIN {X 0,Y 256.041,Z 481.325,A -85,B 0,C 180,E1 -19030.303,E2 -19030.303} C_VEL
LIN {X 0,Y 256.46,Z 477.04,A -85,B 0,C 180,E1 -19032.276,E2 -19032.276} C_VEL
LIN {X 0,Y 255.581,Z 470.55,A -85,B 0,C 180,E1 -19035.639,E2 -19035.639} C_VEL
LIN {X 0,Y 254.289,Z 463.587,A -85,B 0,C 180,E1 -19039.497,E2 -19039.497} C_VEL
LIN {X 0,Y 252.953,Z 457.125,A -85,B 0,C 180,E1 -19043.305,E2 -19043.305} C_VEL
LIN {X 0,Y 251.086,Z 449.843,A -85,B 0,C 180,E1 -19047.871,E2 -19047.871} C_VEL
LIN {X 0,Y 250.794,Z 448.944,A -85,B 0,C 180,E1 -19048.459,E2 -19048.459} C_VEL
LIN {X 0,Y 255.502,Z 463.029,A -85,B 0,C 180,E1 -19050.408,E2 -19050.408} C_VEL
LIN {X 0,Y 259.144,Z 475.546,A -85,B 0,C 180,E1 -19052.304,E2 -19052.304} C_VEL
LIN {X 0,Y 260.034,Z 479.365,A -85,B 0,C 180,E1 -19052.91,E2 -19052.91} C_VEL
LIN {X 0,Y 258.027,Z 492.071,A -85,B 0,C 180,E1 -19054.812,E2 -19054.812} C_VEL
LIN {X 0,Y 255.924,Z 504.13,A -85,B 0,C 180,E1 -19056.963,E2 -19056.963} C_VEL
LIN {X 0,Y 253.988,Z 515.304,A -85,B 0,C 180,E1 -19059.341,E2 -19059.341} C_VEL
LIN {X 0,Y 252.103,Z 526.25,A -85,B 0,C 180,E1 -19062.142,E2 -19062.142} C_VEL
LIN {X 0,Y 250.881,Z 534.198,A -85,B 0,C 180,E1 -19064.566,E2 -19064.566} C_VEL
LIN {X 0,Y 249.719,Z 542.033,A -85,B 0,C 180,E1 -19067.402,E2 -19067.402} C_VEL
LIN {X 0,Y 248.93,Z 548.53,A -85,B 0,C 180,E1 -19070.247,E2 -19070.247} C_VEL
LIN {X 0,Y 248.415,Z 554.518,A -85,B 0,C 180,E1 -19073.502,E2 -19073.502} C_VEL
LIN {X 0,Y 248.191,Z 559.106,A -85,B 0,C 180,E1 -19076.753,E2 -19076.753} C_VEL
LIN {X 0,Y 248.04,Z 562.422,A -85,B 0,C 180,E1 -19080,E2 -19080} C_VEL
LIN {X 0,Y 248.531,Z 564.527,A -85,B 0,C 180,E1 -19083.242,E2 -19083.242} C_VEL
LIN {X 0,Y 249.533,Z 565.462,A -85,B 0,C 180,E1 -19086.468,E2 -19086.468} C_VEL
LIN {X 0,Y 251.156,Z 565.132,A -85,B 0,C 180,E1 -19090.072,E2 -19090.072} C_VEL
LIN {X 0,Y 251.24,Z 564.821,A -85,B 0,C 180,E1 -19091.417,E2 -19091.417} C_VEL
LIN {X 0,Y 249.834,Z 564.281,A -85,B 0,C 180,E1 -19093.66,E2 -19093.66} C_VEL
LIN {X 0,Y 248.799,Z 563.62,A -85,B 0,C 180,E1 -19095.466,E2 -19095.466} C_VEL
LIN {X 0,Y 248.927,Z 562.769,A -85,B 0,C 180,E1 -19096.812,E2 -19096.812} C_VEL
LIN {X 0,Y 249.253,Z 562.371,A -85,B 0,C 180,E1 -19097.251,E2 -19097.251} C_VEL
LIN {X 0,Y 252.663,Z 558.778,A -85,B 0,C 180,E1 -19100.346,E2 -19100.346} C_VEL
LIN {X 0,Y 256.793,Z 553.978,A -85,B 0,C 180,E1 -19103.381,E2 -19103.381} C_VEL
LIN {X 0,Y 261.644,Z 547.916,A -85,B 0,C 180,E1 -19106.308,E2 -19106.308} C_VEL
LIN {X 0,Y 267.288,Z 540.262,A -85,B 0,C 180,E1 -19109.219,E2 -19109.219} C_VEL
LIN {X 0,Y 273.255,Z 531.633,A -85,B 0,C 180,E1 -19111.82,E2 -19111.82} C_VEL
LIN {X 0,Y 280.14,Z 520.994,A -85,B 0,C 180,E1 -19114.365,E2 -19114.365} C_VEL
LIN {X 0,Y 283.76,Z 515.058,A -85,B 0,C 180,E1 -19115.542,E2 -19115.542} C_VEL
LIN {X 0,Y 284.439,Z 513.633,A -85,B 0,C 180,E1 -19115.906,E2 -19115.906} C_VEL
LIN {X 0,Y 284.788,Z 511.403,A -85,B 0,C 180,E1 -19117.069,E2 -19117.069} C_VEL
LIN {X 0,Y 284.416,Z 510.333,A -85,B 0,C 180,E1 -19118.153,E2 -19118.153} C_VEL
LIN {X 0,Y 283.437,Z 509.68,A -85,B 0,C 180,E1 -19120.142,E2 -19120.142} C_VEL
LIN {X 0,Y 282.435,Z 510.235,A -85,B 0,C 180,E1 -19121.711,E2 -19121.711} C_VEL
LIN {X 0,Y 282.037,Z 510.704,A -85,B 0,C 180,E1 -19122.284,E2 -19122.284} C_VEL
LIN {X 0,Y 280.891,Z 512.354,A -85,B 0,C 180,E1 -19123.482,E2 -19123.482} C_VEL
LIN {X 0,Y 278.388,Z 518.069,A -85,B 0,C 180,E1 -19126.498,E2 -19126.498} C_VEL
LIN {X 0,Y 276.599,Z 523.565,A -85,B 0,C 180,E1 -19128.652,E2 -19128.652} C_VEL
LIN {X 0,Y 274.733,Z 530.049,A -85,B 0,C 180,E1 -19130.764,E2 -19130.764} C_VEL
LIN {X 0,Y 272.521,Z 537.289,A -85,B 0,C 180,E1 -19132.789,E2 -19132.789} C_VEL
LIN {X 0,Y 269.767,Z 544.814,A -85,B 0,C 180,E1 -19134.654,E2 -19134.654} C_VEL
LIN {X 0,Y 263.324,Z 559.52,A -85,B 0,C 180,E1 -19138.189,E2 -19138.189} C_VEL
LIN {X 0,Y 261.662,Z 563.627,A -85,B 0,C 180,E1 -19139.315,E2 -19139.315} C_VEL
LIN {X 0,Y 255.749,Z 574.166,A -85,B 0,C 180,E1 -19142.15,E2 -19142.15} C_VEL
LIN {X 0,Y 253.355,Z 578.691,A -85,B 0,C 180,E1 -19143.54,E2 -19143.54} C_VEL
LIN {X 0,Y 250.569,Z 588.523,A -85,B 0,C 180,E1 -19145.562,E2 -19145.562} C_VEL
LIN {X 0,Y 247.934,Z 597.867,A -85,B 0,C 180,E1 -19147.939,E2 -19147.939} C_VEL
LIN {X 0,Y 245.65,Z 605.587,A -85,B 0,C 180,E1 -19150.35,E2 -19150.35} C_VEL
LIN {X 0,Y 243.577,Z 612.993,A -85,B 0,C 180,E1 -19153.23,E2 -19153.23} C_VEL
LIN {X 0,Y 242.131,Z 618.124,A -85,B 0,C 180,E1 -19155.717,E2 -19155.717} C_VEL
LIN {X 0,Y 241.085,Z 622.266,A -85,B 0,C 180,E1 -19158.225,E2 -19158.225} C_VEL
LIN {X 0,Y 240.226,Z 626.44,A -85,B 0,C 180,E1 -19161.589,E2 -19161.589} C_VEL
LIN {X 0,Y 239.841,Z 629.239,A -85,B 0,C 180,E1 -19165.066,E2 -19165.066} C_VEL
LIN {X 0,Y 239.841,Z 630.519,A -85,B 0,C 180,E1 -19168.321,E2 -19168.321} C_VEL
LIN {X 0,Y 239.866,Z 630.686,A -85,B 0,C 180,E1 -19170,E2 -19170} C_VEL
LIN {X 0,Y 239.841,Z 630.513,A -85,B 0,C 180,E1 -19171.679,E2 -19171.679} C_VEL
LIN {X 0,Y 239.844,Z 629.151,A -85,B 0,C 180,E1 -19175.043,E2 -19175.043} C_VEL
LIN {X 0,Y 240.212,Z 626.415,A -85,B 0,C 180,E1 -19178.412,E2 -19178.412} C_VEL
LIN {X 0,Y 241.074,Z 622.225,A -85,B 0,C 180,E1 -19181.775,E2 -19181.775} C_VEL
LIN {X 0,Y 242.106,Z 618.068,A -85,B 0,C 180,E1 -19184.285,E2 -19184.285} C_VEL
LIN {X 0,Y 243.528,Z 612.931,A -85,B 0,C 180,E1 -19186.774,E2 -19186.774} C_VEL
LIN {X 0,Y 245.571,Z 605.525,A -85,B 0,C 180,E1 -19189.65,E2 -19189.65} C_VEL
LIN {X 0,Y 247.882,Z 597.769,A -85,B 0,C 180,E1 -19192.066,E2 -19192.066} C_VEL
LIN {X 0,Y 250.525,Z 588.399,A -85,B 0,C 180,E1 -19194.443,E2 -19194.443} C_VEL
LIN {X 0,Y 253.478,Z 578.006,A -85,B 0,C 180,E1 -19196.557,E2 -19196.557} C_VEL
LIN {X 0,Y 256.019,Z 567.746,A -85,B 0,C 180,E1 -19198.273,E2 -19198.273} C_VEL
LIN {X 0,Y 257.916,Z 558.366,A -85,B 0,C 180,E1 -19199.597,E2 -19199.597} C_VEL
LIN {X 0,Y 257.754,Z 545.959,A -85,B 0,C 180,E1 -19201.335,E2 -19201.335} C_VEL
LIN {X 0,Y 256.979,Z 532.747,A -85,B 0,C 180,E1 -19202.897,E2 -19202.897} C_VEL
LIN {X 0,Y 255.613,Z 519.949,A -85,B 0,C 180,E1 -19204.177,E2 -19204.177} C_VEL
LIN {X 0,Y 252.375,Z 506.842,A -85,B 0,C 180,E1 -19205.471,E2 -19205.471} C_VEL
LIN {X 0,Y 247.372,Z 492.092,A -85,B 0,C 180,E1 -19206.876,E2 -19206.876} C_VEL
LIN {X 0,Y 246.737,Z 490.129,A -85,B 0,C 180,E1 -19207.104,E2 -19207.104} C_VEL
LIN {X 0,Y 245.379,Z 476.807,A -85,B 0,C 180,E1 -19210.626,E2 -19210.626} C_VEL
LIN {X 0,Y 243.952,Z 465.529,A -85,B 0,C 180,E1 -19213.849,E2 -19213.849} C_VEL
LIN {X 0,Y 244.567,Z 460.932,A -85,B 0,C 180,E1 -19217.43,E2 -19217.43} C_VEL
LIN {X 0,Y 244.517,Z 458.066,A -85,B 0,C 180,E1 -19219.707,E2 -19219.707} C_VEL
LIN {X 0,Y 243.65,Z 453.088,A -85,B 0,C 180,E1 -19223.867,E2 -19223.867} C_VEL
LIN {X 0,Y 242.725,Z 447.663,A -85,B 0,C 180,E1 -19228.589,E2 -19228.589} C_VEL
LIN {X 0,Y 242.118,Z 443.944,A -85,B 0,C 180,E1 -19232.091,E2 -19232.091} C_VEL
LIN {X 0,Y 242.059,Z 443.955,A -85,B 0,C 180,E1 -19236.016,E2 -19236.016} C_VEL
LIN {X 0,Y 242.039,Z 443.937,A -85,B 0,C 180,E1 -19239.608,E2 -19239.608} C_VEL
LIN {X 0,Y 242.165,Z 443.936,A -85,B 0,C 180,E1 -19243.278,E2 -19243.278} C_VEL
LIN {X 0,Y 242.181,Z 443.944,A -85,B 0,C 180,E1 -19248.28,E2 -19248.28} C_VEL
LIN {X 0,Y 242.393,Z 443.892,A -85,B 0,C 180,E1 -19251.665,E2 -19251.665} C_VEL
LIN {X 0,Y 242.256,Z 443.928,A -85,B 0,C 180,E1 -19255.007,E2 -19255.007} C_VEL
LIN {X 0,Y 242.638,Z 443.867,A -85,B 0,C 180,E1 -19258.34,E2 -19258.34} C_VEL
LIN {X 0,Y 242.638,Z 443.87,A -85,B 0,C 180,E1 -19261.66,E2 -19261.66} C_VEL
LIN {X 0,Y 242.431,Z 443.905,A -85,B 0,C 180,E1 -19266.732,E2 -19266.732} C_VEL
LIN {X 0,Y 242.316,Z 443.913,A -85,B 0,C 180,E1 -19270.022,E2 -19270.022} C_VEL
LIN {X 0,Y 242.168,Z 443.934,A -85,B 0,C 180,E1 -19275.141,E2 -19275.141} C_VEL
LIN {X 0,Y 242.073,Z 443.941,A -85,B 0,C 180,E1 -19278.624,E2 -19278.624} C_VEL
LIN {X 0,Y 242.008,Z 443.953,A -85,B 0,C 180,E1 -19282.181,E2 -19282.181} C_VEL
LIN {X 0,Y 242.068,Z 444.032,A -85,B 0,C 180,E1 -19285.838,E2 -19285.838} C_VEL
LIN {X 0,Y 243.49,Z 448.819,A -85,B 0,C 180,E1 -19289.386,E2 -19289.386} C_VEL
LIN {X 0,Y 244.932,Z 454.094,A -85,B 0,C 180,E1 -19293.037,E2 -19293.037} C_VEL
LIN {X 0,Y 246.516,Z 460.399,A -85,B 0,C 180,E1 -19297.035,E2 -19297.035} C_VEL
LIN {X 0,Y 247.748,Z 466.535,A -85,B 0,C 180,E1 -19300.727,E2 -19300.727} C_VEL
LIN {X 0,Y 248.759,Z 472.01,A -85,B 0,C 180,E1 -19303.803,E2 -19303.803} C_VEL
LIN {X 0,Y 249.665,Z 478.021,A -85,B 0,C 180,E1 -19307.046,E2 -19307.046} C_VEL
LIN {X 0,Y 249.63,Z 481.125,A -85,B 0,C 180,E1 -19308.578,E2 -19308.578} C_VEL
LIN {X 0,Y 248.304,Z 491.484,A -85,B 0,C 180,E1 -19313.169,E2 -19313.169} C_VEL
LIN {X 0,Y 253.372,Z 506.997,A -85,B 0,C 180,E1 -19314.688,E2 -19314.688} C_VEL
LIN {X 0,Y 256.646,Z 520.836,A -85,B 0,C 180,E1 -19316.152,E2 -19316.152} C_VEL
LIN {X 0,Y 258.834,Z 534.103,A -85,B 0,C 180,E1 -19317.726,E2 -19317.726} C_VEL
LIN {X 0,Y 259.83,Z 546.058,A -85,B 0,C 180,E1 -19319.3,E2 -19319.3} C_VEL
LIN {X 0,Y 259.522,Z 550.905,A -85,B 0,C 180,E1 -19319.935,E2 -19319.935} C_VEL
LIN {X 0,Y 256.86,Z 563.37,A -85,B 0,C 180,E1 -19321.615,E2 -19321.615} C_VEL
LIN {X 0,Y 253.949,Z 574.649,A -85,B 0,C 180,E1 -19323.496,E2 -19323.496} C_VEL
LIN {X 0,Y 251.082,Z 584.885,A -85,B 0,C 180,E1 -19325.615,E2 -19325.615} C_VEL
LIN {X 0,Y 248.364,Z 594.128,A -85,B 0,C 180,E1 -19327.98,E2 -19327.98} C_VEL
LIN {X 0,Y 245.671,Z 602.791,A -85,B 0,C 180,E1 -19330.743,E2 -19330.743} C_VEL
LIN {X 0,Y 244.072,Z 609.118,A -85,B 0,C 180,E1 -19333.265,E2 -19333.265} C_VEL
LIN {X 0,Y 241.994,Z 615.671,A -85,B 0,C 180,E1 -19336.565,E2 -19336.565} C_VEL
LIN {X 0,Y 240.776,Z 620.584,A -85,B 0,C 180,E1 -19339.914,E2 -19339.914} C_VEL
LIN {X 0,Y 240.057,Z 624.005,A -85,B 0,C 180,E1 -19343.275,E2 -19343.275} C_VEL
LIN {X 0,Y 239.79,Z 626.035,A -85,B 0,C 180,E1 -19346.64,E2 -19346.64} C_VEL
LIN {X 0,Y 239.805,Z 626.729,A -85,B 0,C 180,E1 -19350,E2 -19350} C_VEL
LIN {X 0,Y 239.784,Z 626.091,A -85,B 0,C 180,E1 -19353.361,E2 -19353.361} C_VEL
LIN {X 0,Y 240.056,Z 624.105,A -85,B 0,C 180,E1 -19356.725,E2 -19356.725} C_VEL
LIN {X 0,Y 240.771,Z 620.734,A -85,B 0,C 180,E1 -19360.087,E2 -19360.087} C_VEL
LIN {X 0,Y 241.92,Z 615.876,A -85,B 0,C 180,E1 -19363.439,E2 -19363.439} C_VEL
LIN {X 0,Y 244.017,Z 609.376,A -85,B 0,C 180,E1 -19366.739,E2 -19366.739} C_VEL
LIN {X 0,Y 245.871,Z 602.726,A -85,B 0,C 180,E1 -19369.39,E2 -19369.39} C_VEL
LIN {X 0,Y 248.313,Z 594.519,A -85,B 0,C 180,E1 -19372.025,E2 -19372.025} C_VEL
LIN {X 0,Y 250.99,Z 585.374,A -85,B 0,C 180,E1 -19374.395,E2 -19374.395} C_VEL
LIN {X 0,Y 253.859,Z 575.248,A -85,B 0,C 180,E1 -19376.514,E2 -19376.514} C_VEL
LIN {X 0,Y 256.701,Z 564.3,A -85,B 0,C 180,E1 -19378.368,E2 -19378.368} C_VEL
LIN {X 0,Y 259.405,Z 551.779,A -85,B 0,C 180,E1 -19380.08,E2 -19380.08} C_VEL
LIN {X 0,Y 259.98,Z 548.685,A -85,B 0,C 180,E1 -19380.455,E2 -19380.455} C_VEL
LIN {X 0,Y 258.992,Z 535.338,A -85,B 0,C 180,E1 -19382.252,E2 -19382.252} C_VEL
LIN {X 0,Y 256.911,Z 521.825,A -85,B 0,C 180,E1 -19383.86,E2 -19383.86} C_VEL
LIN {X 0,Y 253.646,Z 507.922,A -85,B 0,C 180,E1 -19385.349,E2 -19385.349} C_VEL
LIN {X 0,Y 248.912,Z 493.49,A -85,B 0,C 180,E1 -19386.792,E2 -19386.792} C_VEL
LIN {X 0,Y 248.305,Z 491.21,A -85,B 0,C 180,E1 -19387.034,E2 -19387.034} C_VEL
LIN {X 0,Y 249.628,Z 481.466,A -85,B 0,C 180,E1 -19391.422,E2 -19391.422} C_VEL
LIN {X 0,Y 249.738,Z 478.252,A -85,B 0,C 180,E1 -19392.972,E2 -19392.972} C_VEL
LIN {X 0,Y 248.835,Z 472.238,A -85,B 0,C 180,E1 -19396.214,E2 -19396.214} C_VEL
LIN {X 0,Y 247.448,Z 464.842,A -85,B 0,C 180,E1 -19400.453,E2 -19400.453} C_VEL
LIN {X 0,Y 246.159,Z 458.752,A -85,B 0,C 180,E1 -19404.176,E2 -19404.176} C_VEL
LIN {X 0,Y 244.627,Z 452.547,A -85,B 0,C 180,E1 -19408.353,E2 -19408.353} C_VEL
LIN {X 0,Y 248.968,Z 465.704,A -85,B 0,C 180,E1 -19410.229,E2 -19410.229} C_VEL
LIN {X 0,Y 252.66,Z 478.551,A -85,B 0,C 180,E1 -19412.267,E2 -19412.267} C_VEL
LIN {X 0,Y 253.024,Z 480.973,A -85,B 0,C 180,E1 -19412.661,E2 -19412.661} C_VEL
LIN {X 0,Y 250.887,Z 494.106,A -85,B 0,C 180,E1 -19414.71,E2 -19414.71} C_VEL
LIN {X 0,Y 248.602,Z 506.906,A -85,B 0,C 180,E1 -19417.125,E2 -19417.125} C_VEL
LIN {X 0,Y 246.619,Z 517.728,A -85,B 0,C 180,E1 -19419.568,E2 -19419.568} C_VEL
LIN {X 0,Y 245.028,Z 526.99,A -85,B 0,C 180,E1 -19422.041,E2 -19422.041} C_VEL
LIN {X 0,Y 243.761,Z 534.967,A -85,B 0,C 180,E1 -19424.532,E2 -19424.532} C_VEL
LIN {X 0,Y 242.624,Z 542.834,A -85,B 0,C 180,E1 -19427.452,E2 -19427.452} C_VEL
LIN {X 0,Y 241.697,Z 550.324,A -85,B 0,C 180,E1 -19430.882,E2 -19430.882} C_VEL
LIN {X 0,Y 241.273,Z 555.961,A -85,B 0,C 180,E1 -19434.148,E2 -19434.148} C_VEL
LIN {X 0,Y 241.107,Z 559.412,A -85,B 0,C 180,E1 -19436.658,E2 -19436.658} C_VEL
LIN {X 0,Y 240.977,Z 562.93,A -85,B 0,C 180,E1 -19440,E2 -19440} C_VEL
LIN {X 0,Y 241.489,Z 565.23,A -85,B 0,C 180,E1 -19443.337,E2 -19443.337} C_VEL
LIN {X 0,Y 242.551,Z 566.364,A -85,B 0,C 180,E1 -19446.656,E2 -19446.656} C_VEL
LIN {X 0,Y 244.226,Z 566.295,A -85,B 0,C 180,E1 -19450.283,E2 -19450.283} C_VEL
LIN {X 0,Y 246.003,Z 565.304,A -85,B 0,C 180,E1 -19453.212,E2 -19453.212} C_VEL
LIN {X 0,Y 248.501,Z 563.15,A -85,B 0,C 180,E1 -19456.428,E2 -19456.428} C_VEL
LIN {X 0,Y 249.253,Z 562.371,A -85,B 0,C 180,E1 -19457.251,E2 -19457.251} C_VEL
LIN {X 0,Y 249.935,Z 561.263,A -85,B 0,C 180,E1 -19458.576,E2 -19458.576} C_VEL
LIN {X 0,Y 249.673,Z 558.011,A -85,B 0,C 180,E1 -19462.601,E2 -19462.601} C_VEL
LIN {X 0,Y 250.541,Z 556.349,A -85,B 0,C 180,E1 -19463.88,E2 -19463.88} C_VEL
LIN {X 0,Y 251.097,Z 555.676,A -85,B 0,C 180,E1 -19464.281,E2 -19464.281} C_VEL
LIN {X 0,Y 255.723,Z 550.458,A -85,B 0,C 180,E1 -19466.966,E2 -19466.966} C_VEL
LIN {X 0,Y 261.435,Z 543.476,A -85,B 0,C 180,E1 -19469.823,E2 -19469.823} C_VEL
LIN {X 0,Y 267.487,Z 535.587,A -85,B 0,C 180,E1 -19472.399,E2 -19472.399} C_VEL
LIN {X 0,Y 274.087,Z 526.412,A -85,B 0,C 180,E1 -19474.787,E2 -19474.787} C_VEL
LIN {X 0,Y 279.814,Z 517.918,A -85,B 0,C 180,E1 -19476.621,E2 -19476.621} C_VEL
LIN {X 0,Y 279.981,Z 517.139,A -85,B 0,C 180,E1 -19477.045,E2 -19477.045} C_VEL
LIN {X 0,Y 279.581,Z 515.59,A -85,B 0,C 180,E1 -19478.935,E2 -19478.935} C_VEL
LIN {X 0,Y 278.465,Z 515.63,A -85,B 0,C 180,E1 -19481.011,E2 -19481.011} C_VEL
LIN {X 0,Y 277.121,Z 517.153,A -85,B 0,C 180,E1 -19482.654,E2 -19482.654} C_VEL
LIN {X 0,Y 273.806,Z 523.418,A -85,B 0,C 180,E1 -19486.129,E2 -19486.129} C_VEL
LIN {X 0,Y 271.744,Z 528.658,A -85,B 0,C 180,E1 -19488.266,E2 -19488.266} C_VEL
LIN {X 0,Y 269.23,Z 535.648,A -85,B 0,C 180,E1 -19490.593,E2 -19490.593} C_VEL
LIN {X 0,Y 266.048,Z 543.77,A -85,B 0,C 180,E1 -19492.885,E2 -19492.885} C_VEL
LIN {X 0,Y 262.353,Z 551.58,A -85,B 0,C 180,E1 -19494.834,E2 -19494.834} C_VEL
LIN {X 0,Y 257.465,Z 561.46,A -85,B 0,C 180,E1 -19497.423,E2 -19497.423} C_VEL
LIN {X 0,Y 255.709,Z 565.267,A -85,B 0,C 180,E1 -19498.52,E2 -19498.52} C_VEL
LIN {X 0,Y 249.568,Z 575.265,A -85,B 0,C 180,E1 -19501.397,E2 -19501.397} C_VEL
LIN {X 0,Y 246.409,Z 580.632,A -85,B 0,C 180,E1 -19503.192,E2 -19503.192} C_VEL
LIN {X 0,Y 243.627,Z 590.134,A -85,B 0,C 180,E1 -19505.273,E2 -19505.273} C_VEL
LIN {X 0,Y 240.879,Z 599.172,A -85,B 0,C 180,E1 -19507.71,E2 -19507.71} C_VEL
LIN {X 0,Y 238.527,Z 606.906,A -85,B 0,C 180,E1 -19510.284,E2 -19510.284} C_VEL
LIN {X 0,Y 236.752,Z 612.938,A -85,B 0,C 180,E1 -19512.731,E2 -19512.731} C_VEL
LIN {X 0,Y 235.229,Z 618.068,A -85,B 0,C 180,E1 -19515.288,E2 -19515.288} C_VEL
LIN {X 0,Y 234.095,Z 622.209,A -85,B 0,C 180,E1 -19517.869,E2 -19517.869} C_VEL
LIN {X 0,Y 233.188,Z 626.382,A -85,B 0,C 180,E1 -19521.333,E2 -19521.333} C_VEL
LIN {X 0,Y 232.767,Z 629.108,A -85,B 0,C 180,E1 -19524.803,E2 -19524.803} C_VEL
LIN {X 0,Y 232.754,Z 630.461,A -85,B 0,C 180,E1 -19528.27,E2 -19528.27} C_VEL
LIN {X 0,Y 232.778,Z 630.627,A -85,B 0,C 180,E1 -19530,E2 -19530} C_VEL
LIN {X 0,Y 232.753,Z 630.454,A -85,B 0,C 180,E1 -19531.73,E2 -19531.73} C_VEL
LIN {X 0,Y 232.767,Z 629.092,A -85,B 0,C 180,E1 -19535.197,E2 -19535.197} C_VEL
LIN {X 0,Y 233.177,Z 626.356,A -85,B 0,C 180,E1 -19538.668,E2 -19538.668} C_VEL
LIN {X 0,Y 234.084,Z 622.166,A -85,B 0,C 180,E1 -19542.132,E2 -19542.132} C_VEL
LIN {X 0,Y 235.205,Z 618.009,A -85,B 0,C 180,E1 -19544.713,E2 -19544.713} C_VEL
LIN {X 0,Y 236.699,Z 612.873,A -85,B 0,C 180,E1 -19547.273,E2 -19547.273} C_VEL
LIN {X 0,Y 238.855,Z 605.468,A -85,B 0,C 180,E1 -19550.226,E2 -19550.226} C_VEL
LIN {X 0,Y 241.282,Z 597.712,A -85,B 0,C 180,E1 -19552.702,E2 -19552.702} C_VEL
LIN {X 0,Y 244.053,Z 588.345,A -85,B 0,C 180,E1 -19555.135,E2 -19555.135} C_VEL
LIN {X 0,Y 247.129,Z 577.953,A -85,B 0,C 180,E1 -19557.295,E2 -19557.295} C_VEL
LIN {X 0,Y 249.984,Z 566.668,A -85,B 0,C 180,E1 -19559.205,E2 -19559.205} C_VEL
LIN {X 0,Y 251.477,Z 559.735,A -85,B 0,C 180,E1 -19560.202,E2 -19560.202} C_VEL
LIN {X 0,Y 251.482,Z 548.687,A -85,B 0,C 180,E1 -19561.836,E2 -19561.836} C_VEL
LIN {X 0,Y 250.91,Z 534.913,A -85,B 0,C 180,E1 -19563.567,E2 -19563.567} C_VEL
LIN {X 0,Y 249.747,Z 522.39,A -85,B 0,C 180,E1 -19564.899,E2 -19564.899} C_VEL
LIN {X 0,Y 246.767,Z 509.559,A -85,B 0,C 180,E1 -19566.255,E2 -19566.255} C_VEL
LIN {X 0,Y 242.164,Z 495.451,A -85,B 0,C 180,E1 -19567.684,E2 -19567.684} C_VEL
LIN {X 0,Y 240.256,Z 490.093,A -85,B 0,C 180,E1 -19568.301,E2 -19568.301} C_VEL
LIN {X 0,Y 239.15,Z 478.83,A -85,B 0,C 180,E1 -19571.465,E2 -19571.465} C_VEL
LIN {X 0,Y 238.169,Z 469.606,A -85,B 0,C 180,E1 -19574.174,E2 -19574.174} C_VEL
LIN {X 0,Y 237.347,Z 463.415,A -85,B 0,C 180,E1 -19576.133,E2 -19576.133} C_VEL
LIN {X 0,Y 237.362,Z 462.541,A -85,B 0,C 180,E1 -19576.609,E2 -19576.609} C_VEL
LIN {X 0,Y 237.484,Z 459.123,A -85,B 0,C 180,E1 -19579.379,E2 -19579.379} C_VEL
LIN {X 0,Y 236.726,Z 454.56,A -85,B 0,C 180,E1 -19583.282,E2 -19583.282} C_VEL
LIN {X 0,Y 235.855,Z 449.719,A -85,B 0,C 180,E1 -19587.564,E2 -19587.564} C_VEL
LIN {X 0,Y 235.224,Z 445.51,A -85,B 0,C 180,E1 -19591.442,E2 -19591.442} C_VEL
LIN {X 0,Y 235.064,Z 444.821,A -85,B 0,C 180,E1 -19592.15,E2 -19592.15} C_VEL
LIN {X 0,Y 234.963,Z 444.84,A -85,B 0,C 180,E1 -19597.117,E2 -19597.117} C_VEL
LIN {X 0,Y 235.01,Z 444.82,A -85,B 0,C 180,E1 -19600.795,E2 -19600.795} C_VEL
LIN {X 0,Y 235.115,Z 444.8,A -85,B 0,C 180,E1 -19604.394,E2 -19604.394} C_VEL
LIN {X 0,Y 235.215,Z 444.793,A -85,B 0,C 180,E1 -19609.673,E2 -19609.673} C_VEL
LIN {X 0,Y 235.368,Z 444.784,A -85,B 0,C 180,E1 -19613.14,E2 -19613.14} C_VEL
LIN {X 0,Y 235.597,Z 444.743,A -85,B 0,C 180,E1 -19618.291,E2 -19618.291} C_VEL
LIN {X 0,Y 235.597,Z 444.745,A -85,B 0,C 180,E1 -19621.71,E2 -19621.71} C_VEL
LIN {X 0,Y 235.406,Z 444.777,A -85,B 0,C 180,E1 -19626.859,E2 -19626.859} C_VEL
LIN {X 0,Y 235.24,Z 444.798,A -85,B 0,C 180,E1 -19630.327,E2 -19630.327} C_VEL
LIN {X 0,Y 235.115,Z 444.818,A -85,B 0,C 180,E1 -19635.606,E2 -19635.606} C_VEL
LIN {X 0,Y 235.009,Z 444.822,A -85,B 0,C 180,E1 -19639.206,E2 -19639.206} C_VEL
LIN {X 0,Y 235.028,Z 445.013,A -85,B 0,C 180,E1 -19643.809,E2 -19643.809} C_VEL
LIN {X 0,Y 236.499,Z 449.58,A -85,B 0,C 180,E1 -19647.426,E2 -19647.426} C_VEL
LIN {X 0,Y 238.295,Z 455.952,A -85,B 0,C 180,E1 -19652.065,E2 -19652.065} C_VEL
LIN {X 0,Y 239.678,Z 461.712,A -85,B 0,C 180,E1 -19655.906,E2 -19655.906} C_VEL
LIN {X 0,Y 240.696,Z 466.452,A -85,B 0,C 180,E1 -19658.886,E2 -19658.886} C_VEL
LIN {X 0,Y 241.995,Z 473.535,A -85,B 0,C 180,E1 -19663.091,E2 -19663.091} C_VEL
LIN {X 0,Y 242.917,Z 479.364,A -85,B 0,C 180,E1 -19666.327,E2 -19666.327} C_VEL
LIN {X 0,Y 242.957,Z 483.247,A -85,B 0,C 180,E1 -19668.293,E2 -19668.293} C_VEL
LIN {X 0,Y 241.814,Z 491.464,A -85,B 0,C 180,E1 -19672.01,E2 -19672.01} C_VEL
LIN {X 0,Y 247.063,Z 507.348,A -85,B 0,C 180,E1 -19673.666,E2 -19673.666} C_VEL
LIN {X 0,Y 250.298,Z 520.863,A -85,B 0,C 180,E1 -19675.172,E2 -19675.172} C_VEL
LIN {X 0,Y 252.462,Z 534.366,A -85,B 0,C 180,E1 -19676.832,E2 -19676.832} C_VEL
LIN {X 0,Y 253.451,Z 546.103,A -85,B 0,C 180,E1 -19678.44,E2 -19678.44} C_VEL
LIN {X 0,Y 253.386,Z 550.951,A -85,B 0,C 180,E1 -19679.129,E2 -19679.129} C_VEL
LIN {X 0,Y 250.622,Z 563.42,A -85,B 0,C 180,E1 -19680.841,E2 -19680.841} C_VEL
LIN {X 0,Y 247.6,Z 574.702,A -85,B 0,C 180,E1 -19682.761,E2 -19682.761} C_VEL
LIN {X 0,Y 244.606,Z 584.94,A -85,B 0,C 180,E1 -19684.926,E2 -19684.926} C_VEL
LIN {X 0,Y 241.787,Z 594.184,A -85,B 0,C 180,E1 -19687.348,E2 -19687.348} C_VEL
LIN {X 0,Y 239.063,Z 602.538,A -85,B 0,C 180,E1 -19690.062,E2 -19690.062} C_VEL
LIN {X 0,Y 237.258,Z 609.176,A -85,B 0,C 180,E1 -19692.769,E2 -19692.769} C_VEL
LIN {X 0,Y 235.058,Z 615.73,A -85,B 0,C 180,E1 -19696.161,E2 -19696.161} C_VEL
LIN {X 0,Y 233.761,Z 620.643,A -85,B 0,C 180,E1 -19699.608,E2 -19699.608} C_VEL
LIN {X 0,Y 232.997,Z 624.064,A -85,B 0,C 180,E1 -19703.07,E2 -19703.07} C_VEL
LIN {X 0,Y 232.702,Z 626.094,A -85,B 0,C 180,E1 -19706.537,E2 -19706.537} C_VEL
LIN {X 0,Y 232.72,Z 626.788,A -85,B 0,C 180,E1 -19710,E2 -19710} C_VEL
LIN {X 0,Y 232.696,Z 626.149,A -85,B 0,C 180,E1 -19713.463,E2 -19713.463} C_VEL
LIN {X 0,Y 232.996,Z 624.163,A -85,B 0,C 180,E1 -19716.93,E2 -19716.93} C_VEL
LIN {X 0,Y 233.753,Z 620.791,A -85,B 0,C 180,E1 -19720.393,E2 -19720.393} C_VEL
LIN {X 0,Y 234.983,Z 615.933,A -85,B 0,C 180,E1 -19723.843,E2 -19723.843} C_VEL
LIN {X 0,Y 237.192,Z 609.431,A -85,B 0,C 180,E1 -19727.235,E2 -19727.235} C_VEL
LIN {X 0,Y 239.185,Z 602.681,A -85,B 0,C 180,E1 -19729.995,E2 -19729.995} C_VEL
LIN {X 0,Y 241.713,Z 594.571,A -85,B 0,C 180,E1 -19732.66,E2 -19732.66} C_VEL
LIN {X 0,Y 244.521,Z 585.423,A -85,B 0,C 180,E1 -19735.084,E2 -19735.084} C_VEL
LIN {X 0,Y 247.501,Z 575.294,A -85,B 0,C 180,E1 -19737.251,E2 -19737.251} C_VEL
LIN {X 0,Y 250.683,Z 563.466,A -85,B 0,C 180,E1 -19739.272,E2 -19739.272} C_VEL
LIN {X 0,Y 253.27,Z 551.814,A -85,B 0,C 180,E1 -19740.887,E2 -19740.887} C_VEL
LIN {X 0,Y 253.626,Z 548.721,A -85,B 0,C 180,E1 -19741.303,E2 -19741.303} C_VEL
LIN {X 0,Y 252.799,Z 536.899,A -85,B 0,C 180,E1 -19742.964,E2 -19742.964} C_VEL
LIN {X 0,Y 250.988,Z 524.206,A -85,B 0,C 180,E1 -19744.566,E2 -19744.566} C_VEL
LIN {X 0,Y 247.98,Z 510.533,A -85,B 0,C 180,E1 -19746.128,E2 -19746.128} C_VEL
LIN {X 0,Y 243.786,Z 497.102,A -85,B 0,C 180,E1 -19747.559,E2 -19747.559} C_VEL
LIN {X 0,Y 241.853,Z 491.24,A -85,B 0,C 180,E1 -19748.178,E2 -19748.178} C_VEL
LIN {X 0,Y 243.074,Z 482.45,A -85,B 0,C 180,E1 -19752.239,E2 -19752.239} C_VEL
LIN {X 0,Y 242.905,Z 479.065,A -85,B 0,C 180,E1 -19753.979,E2 -19753.979} C_VEL
LIN {X 0,Y 241.747,Z 471.853,A -85,B 0,C 180,E1 -19758.037,E2 -19758.037} C_VEL
LIN {X 0,Y 240.455,Z 465.075,A -85,B 0,C 180,E1 -19762.136,E2 -19762.136} C_VEL
LIN {X 0,Y 239.335,Z 460.095,A -85,B 0,C 180,E1 -19765.307,E2 -19765.307} C_VEL
LIN {X 0,Y 238.405,Z 456.013,A -85,B 0,C 180,E1 -19768.22,E2 -19768.22} C_VEL
LIN {X 0,Y 242.367,Z 468.125,A -85,B 0,C 180,E1 -19770.041,E2 -19770.041} C_VEL
LIN {X 0,Y 246.119,Z 481.6,A -85,B 0,C 180,E1 -19772.278,E2 -19772.278} C_VEL
LIN {X 0,Y 243.69,Z 495.896,A -85,B 0,C 180,E1 -19774.596,E2 -19774.596} C_VEL
LIN {X 0,Y 241.59,Z 507.582,A -85,B 0,C 180,E1 -19776.876,E2 -19776.876} C_VEL
LIN {X 0,Y 239.318,Z 519.716,A -85,B 0,C 180,E1 -19779.71,E2 -19779.71} C_VEL
LIN {X 0,Y 237.802,Z 529.158,A -85,B 0,C 180,E1 -19782.366,E2 -19782.366} C_VEL
LIN {X 0,Y 236.274,Z 538.098,A -85,B 0,C 180,E1 -19785.355,E2 -19785.355} C_VEL
LIN {X 0,Y 235.357,Z 544.561,A -85,B 0,C 180,E1 -19787.934,E2 -19787.934} C_VEL
LIN {X 0,Y 234.523,Z 551.852,A -85,B 0,C 180,E1 -19791.462,E2 -19791.462} C_VEL
LIN {X 0,Y 234.152,Z 557.381,A -85,B 0,C 180,E1 -19794.834,E2 -19794.834} C_VEL
LIN {X 0,Y 233.968,Z 561.716,A -85,B 0,C 180,E1 -19798.279,E2 -19798.279} C_VEL
LIN {X 0,Y 234.105,Z 564.815,A -85,B 0,C 180,E1 -19801.72,E2 -19801.72} C_VEL
LIN {X 0,Y 234.948,Z 566.732,A -85,B 0,C 180,E1 -19805.148,E2 -19805.148} C_VEL
LIN {X 0,Y 236.303,Z 567.518,A -85,B 0,C 180,E1 -19808.552,E2 -19808.552} C_VEL
LIN {X 0,Y 238.136,Z 567.173,A -85,B 0,C 180,E1 -19811.922,E2 -19811.922} C_VEL
LIN {X 0,Y 240.604,Z 565.672,A -85,B 0,C 180,E1 -19815.436,E2 -19815.436} C_VEL
LIN {X 0,Y 243.445,Z 563.277,A -85,B 0,C 180,E1 -19818.515,E2 -19818.515} C_VEL
LIN {X 0,Y 247.305,Z 559.637,A -85,B 0,C 180,E1 -19821.681,E2 -19821.681} C_VEL
LIN {X 0,Y 251.097,Z 555.676,A -85,B 0,C 180,E1 -19824.281,E2 -19824.281} C_VEL
LIN {X 0,Y 252.488,Z 553.768,A -85,B 0,C 180,E1 -19825.512,E2 -19825.512} C_VEL
LIN {X 0,Y 254.393,Z 548.632,A -85,B 0,C 180,E1 -19829.354,E2 -19829.354} C_VEL
LIN {X 0,Y 255.858,Z 546.409,A -85,B 0,C 180,E1 -19830.535,E2 -19830.535} C_VEL
LIN {X 0,Y 256.58,Z 545.538,A -85,B 0,C 180,E1 -19830.894,E2 -19830.894} C_VEL
LIN {X 0,Y 263.395,Z 537.488,A -85,B 0,C 180,E1 -19833.618,E2 -19833.618} C_VEL
LIN {X 0,Y 271.919,Z 526.51,A -85,B 0,C 180,E1 -19836.474,E2 -19836.474} C_VEL
LIN {X 0,Y 274.184,Z 523.447,A -85,B 0,C 180,E1 -19837.131,E2 -19837.131} C_VEL
LIN {X 0,Y 275.08,Z 521.952,A -85,B 0,C 180,E1 -19837.625,E2 -19837.625} C_VEL
LIN {X 0,Y 274.49,Z 520.996,A -85,B 0,C 180,E1 -19839.815,E2 -19839.815} C_VEL
LIN {X 0,Y 272.975,Z 522.208,A -85,B 0,C 180,E1 -19842.02,E2 -19842.02} C_VEL
LIN {X 0,Y 269.597,Z 527.535,A -85,B 0,C 180,E1 -19845.263,E2 -19845.263} C_VEL
LIN {X 0,Y 266.769,Z 533.517,A -85,B 0,C 180,E1 -19847.826,E2 -19847.826} C_VEL
LIN {X 0,Y 263.688,Z 540.546,A -85,B 0,C 180,E1 -19850.233,E2 -19850.233} C_VEL
LIN {X 0,Y 260.309,Z 547.718,A -85,B 0,C 180,E1 -19852.336,E2 -19852.336} C_VEL
LIN {X 0,Y 253.85,Z 559.309,A -85,B 0,C 180,E1 -19855.42,E2 -19855.42} C_VEL
LIN {X 0,Y 249.826,Z 566.854,A -85,B 0,C 180,E1 -19857.69,E2 -19857.69} C_VEL
LIN {X 0,Y 243.432,Z 576.339,A -85,B 0,C 180,E1 -19860.607,E2 -19860.607} C_VEL
LIN {X 0,Y 239.487,Z 582.534,A -85,B 0,C 180,E1 -19862.826,E2 -19862.826} C_VEL
LIN {X 0,Y 236.666,Z 591.705,A -85,B 0,C 180,E1 -19864.965,E2 -19864.965} C_VEL
LIN {X 0,Y 233.846,Z 600.469,A -85,B 0,C 180,E1 -19867.469,E2 -19867.469} C_VEL
LIN {X 0,Y 231.177,Z 608.855,A -85,B 0,C 180,E1 -19870.463,E2 -19870.463} C_VEL
LIN {X 0,Y 229.389,Z 614.688,A -85,B 0,C 180,E1 -19873.079,E2 -19873.079} C_VEL
LIN {X 0,Y 227.834,Z 619.484,A -85,B 0,C 180,E1 -19875.713,E2 -19875.713} C_VEL
LIN {X 0,Y 226.556,Z 624.426,A -85,B 0,C 180,E1 -19879.273,E2 -19879.273} C_VEL
LIN {X 0,Y 225.842,Z 627.862,A -85,B 0,C 180,E1 -19882.849,E2 -19882.849} C_VEL
LIN {X 0,Y 225.623,Z 629.896,A -85,B 0,C 180,E1 -19886.428,E2 -19886.428} C_VEL
LIN {X 0,Y 225.692,Z 630.569,A -85,B 0,C 180,E1 -19890,E2 -19890} C_VEL
LIN {X 0,Y 225.621,Z 629.883,A -85,B 0,C 180,E1 -19893.572,E2 -19893.572} C_VEL
LIN {X 0,Y 225.838,Z 627.84,A -85,B 0,C 180,E1 -19897.151,E2 -19897.151} C_VEL
LIN {X 0,Y 226.543,Z 624.391,A -85,B 0,C 180,E1 -19900.727,E2 -19900.727} C_VEL
LIN {X 0,Y 227.812,Z 619.43,A -85,B 0,C 180,E1 -19904.288,E2 -19904.288} C_VEL
LIN {X 0,Y 229.349,Z 614.62,A -85,B 0,C 180,E1 -19906.925,E2 -19906.925} C_VEL
LIN {X 0,Y 231.443,Z 607.66,A -85,B 0,C 180,E1 -19909.975,E2 -19909.975} C_VEL
LIN {X 0,Y 234.256,Z 599.018,A -85,B 0,C 180,E1 -19912.956,E2 -19912.956} C_VEL
LIN {X 0,Y 237.098,Z 589.961,A -85,B 0,C 180,E1 -19915.455,E2 -19915.455} C_VEL
LIN {X 0,Y 239.881,Z 580.92,A -85,B 0,C 180,E1 -19917.48,E2 -19917.48} C_VEL
LIN {X 0,Y 242.908,Z 570.116,A -85,B 0,C 180,E1 -19919.463,E2 -19919.463} C_VEL
LIN {X 0,Y 245.111,Z 560.716,A -85,B 0,C 180,E1 -19920.898,E2 -19920.898} C_VEL
LIN {X 0,Y 245.229,Z 548.643,A -85,B 0,C 180,E1 -19922.748,E2 -19922.748} C_VEL
LIN {X 0,Y 244.792,Z 535.327,A -85,B 0,C 180,E1 -19924.472,E2 -19924.472} C_VEL
LIN {X 0,Y 243.847,Z 524.244,A -85,B 0,C 180,E1 -19925.713,E2 -19925.713} C_VEL
LIN {X 0,Y 240.775,Z 510.607,A -85,B 0,C 180,E1 -19927.246,E2 -19927.246} C_VEL
LIN {X 0,Y 236.122,Z 496.449,A -85,B 0,C 180,E1 -19928.79,E2 -19928.79} C_VEL
LIN {X 0,Y 233.816,Z 490.283,A -85,B 0,C 180,E1 -19929.524,E2 -19929.524} C_VEL
LIN {X 0,Y 232.94,Z 478.816,A -85,B 0,C 180,E1 -19932.92,E2 -19932.92} C_VEL
LIN {X 0,Y 231.705,Z 467.038,A -85,B 0,C 180,E1 -19936.716,E2 -19936.716} C_VEL
LIN {X 0,Y 230.39,Z 459.513,A -85,B 0,C 180,E1 -19939.609,E2 -19939.609} C_VEL
LIN {X 0,Y 229.809,Z 455.984,A -85,B 0,C 180,E1 -19942.668,E2 -19942.668} C_VEL
LIN {X 0,Y 228.834,Z 450.672,A -85,B 0,C 180,E1 -19947.489,E2 -19947.489} C_VEL
LIN {X 0,Y 228.18,Z 446.428,A -85,B 0,C 180,E1 -19951.484,E2 -19951.484} C_VEL
LIN {X 0,Y 228.008,Z 445.695,A -85,B 0,C 180,E1 -19952.461,E2 -19952.461} C_VEL
LIN {X 0,Y 227.931,Z 445.706,A -85,B 0,C 180,E1 -19957.671,E2 -19957.671} C_VEL
LIN {X 0,Y 228.036,Z 445.702,A -85,B 0,C 180,E1 -19962.826,E2 -19962.826} C_VEL
LIN {X 0,Y 228.073,Z 445.697,A -85,B 0,C 180,E1 -19967.543,E2 -19967.543} C_VEL
LIN {X 0,Y 228.263,Z 445.649,A -85,B 0,C 180,E1 -19971.145,E2 -19971.145} C_VEL
LIN {X 0,Y 228.319,Z 445.657,A -85,B 0,C 180,E1 -19972.928,E2 -19972.928} C_VEL
LIN {X 0,Y 228.556,Z 445.619,A -85,B 0,C 180,E1 -19978.238,E2 -19978.238} C_VEL
LIN {X 0,Y 228.556,Z 445.621,A -85,B 0,C 180,E1 -19981.762,E2 -19981.762} C_VEL
LIN {X 0,Y 228.357,Z 445.651,A -85,B 0,C 180,E1 -19987.072,E2 -19987.072} C_VEL
LIN {X 0,Y 228.165,Z 445.684,A -85,B 0,C 180,E1 -19990.65,E2 -19990.65} C_VEL
LIN {X 0,Y 228.066,Z 445.682,A -85,B 0,C 180,E1 -19994.272,E2 -19994.272} C_VEL
LIN {X 0,Y 228.004,Z 445.694,A -85,B 0,C 180,E1 -19997.953,E2 -19997.953} C_VEL
LIN {X 0,Y 227.953,Z 445.753,A -85,B 0,C 180,E1 -20001.239,E2 -20001.239} C_VEL
LIN {X 0,Y 229.5,Z 450.573,A -85,B 0,C 180,E1 -20005.387,E2 -20005.387} C_VEL
LIN {X 0,Y 230.893,Z 455.221,A -85,B 0,C 180,E1 -20009.145,E2 -20009.145} C_VEL
LIN {X 0,Y 232.299,Z 460.591,A -85,B 0,C 180,E1 -20012.996,E2 -20012.996} C_VEL
LIN {X 0,Y 233.664,Z 466.43,A -85,B 0,C 180,E1 -20016.981,E2 -20016.981} C_VEL
LIN {X 0,Y 235.076,Z 473.934,A -85,B 0,C 180,E1 -20021.633,E2 -20021.633} C_VEL
LIN {X 0,Y 236.138,Z 480.805,A -85,B 0,C 180,E1 -20025.586,E2 -20025.586} C_VEL
LIN {X 0,Y 236.416,Z 484.64,A -85,B 0,C 180,E1 -20027.63,E2 -20027.63} C_VEL
LIN {X 0,Y 235.4,Z 491.376,A -85,B 0,C 180,E1 -20030.779,E2 -20030.779} C_VEL
LIN {X 0,Y 240.504,Z 506.747,A -85,B 0,C 180,E1 -20032.471,E2 -20032.471} C_VEL
LIN {X 0,Y 243.506,Z 518.578,A -85,B 0,C 180,E1 -20033.85,E2 -20033.85} C_VEL
LIN {X 0,Y 245.772,Z 531.512,A -85,B 0,C 180,E1 -20035.479,E2 -20035.479} C_VEL
LIN {X 0,Y 246.94,Z 542.962,A -85,B 0,C 180,E1 -20037.059,E2 -20037.059} C_VEL
LIN {X 0,Y 247.216,Z 550.997,A -85,B 0,C 180,E1 -20038.27,E2 -20038.27} C_VEL
LIN {X 0,Y 244.386,Z 563.718,A -85,B 0,C 180,E1 -20040.069,E2 -20040.069} C_VEL
LIN {X 0,Y 241.289,Z 574.754,A -85,B 0,C 180,E1 -20041.987,E2 -20041.987} C_VEL
LIN {X 0,Y 238.185,Z 584.995,A -85,B 0,C 180,E1 -20044.201,E2 -20044.201} C_VEL
LIN {X 0,Y 235.225,Z 594.241,A -85,B 0,C 180,E1 -20046.679,E2 -20046.679} C_VEL
LIN {X 0,Y 232.281,Z 602.857,A -85,B 0,C 180,E1 -20049.564,E2 -20049.564} C_VEL
LIN {X 0,Y 230.448,Z 609.235,A -85,B 0,C 180,E1 -20052.244,E2 -20052.244} C_VEL
LIN {X 0,Y 228.135,Z 615.789,A -85,B 0,C 180,E1 -20055.732,E2 -20055.732} C_VEL
LIN {X 0,Y 226.762,Z 620.702,A -85,B 0,C 180,E1 -20059.283,E2 -20059.283} C_VEL
LIN {X 0,Y 225.935,Z 624.123,A -85,B 0,C 180,E1 -20062.852,E2 -20062.852} C_VEL
LIN {X 0,Y 225.616,Z 626.153,A -85,B 0,C 180,E1 -20066.428,E2 -20066.428} C_VEL
LIN {X 0,Y 225.636,Z 626.846,A -85,B 0,C 180,E1 -20070,E2 -20070} C_VEL
LIN {X 0,Y 225.611,Z 626.207,A -85,B 0,C 180,E1 -20073.572,E2 -20073.572} C_VEL
LIN {X 0,Y 225.934,Z 624.221,A -85,B 0,C 180,E1 -20077.148,E2 -20077.148} C_VEL
LIN {X 0,Y 226.753,Z 620.848,A -85,B 0,C 180,E1 -20080.717,E2 -20080.717} C_VEL
LIN {X 0,Y 228.061,Z 615.989,A -85,B 0,C 180,E1 -20084.272,E2 -20084.272} C_VEL
LIN {X 0,Y 230.362,Z 609.487,A -85,B 0,C 180,E1 -20087.763,E2 -20087.763} C_VEL
LIN {X 0,Y 232.4,Z 602.954,A -85,B 0,C 180,E1 -20090.513,E2 -20090.513} C_VEL
LIN {X 0,Y 235.158,Z 594.623,A -85,B 0,C 180,E1 -20093.328,E2 -20093.328} C_VEL
LIN {X 0,Y 238.098,Z 585.473,A -85,B 0,C 180,E1 -20095.81,E2 -20095.81} C_VEL
LIN {X 0,Y 241.182,Z 575.34,A -85,B 0,C 180,E1 -20098.026,E2 -20098.026} C_VEL
LIN {X 0,Y 244.413,Z 563.856,A -85,B 0,C 180,E1 -20100.034,E2 -20100.034} C_VEL
LIN {X 0,Y 247.185,Z 551.843,A -85,B 0,C 180,E1 -20101.735,E2 -20101.735} C_VEL
LIN {X 0,Y 246.919,Z 541.854,A -85,B 0,C 180,E1 -20103.229,E2 -20103.229} C_VEL
LIN {X 0,Y 245.527,Z 529.469,A -85,B 0,C 180,E1 -20104.924,E2 -20104.924} C_VEL
LIN {X 0,Y 243.031,Z 516.151,A -85,B 0,C 180,E1 -20106.57,E2 -20106.57} C_VEL
LIN {X 0,Y 239.424,Z 503.122,A -85,B 0,C 180,E1 -20108.08,E2 -20108.08} C_VEL
LIN {X 0,Y 235.439,Z 491.248,A -85,B 0,C 180,E1 -20109.404,E2 -20109.404} C_VEL
LIN {X 0,Y 236.385,Z 484.939,A -85,B 0,C 180,E1 -20112.374,E2 -20112.374} C_VEL
LIN {X 0,Y 236.222,Z 481.051,A -85,B 0,C 180,E1 -20114.435,E2 -20114.435} C_VEL
LIN {X 0,Y 235.16,Z 474.289,A -85,B 0,C 180,E1 -20118.344,E2 -20118.344} C_VEL
LIN {X 0,Y 233.769,Z 466.693,A -85,B 0,C 180,E1 -20123.038,E2 -20123.038} C_VEL
LIN {X 0,Y 232.342,Z 460.843,A -85,B 0,C 180,E1 -20127.011,E2 -20127.011} C_VEL
LIN {X 0,Y 232.096,Z 459.4,A -85,B 0,C 180,E1 -20128.081,E2 -20128.081} C_VEL
LIN {X 0,Y 235.365,Z 469.215,A -85,B 0,C 180,E1 -20129.633,E2 -20129.633} C_VEL
LIN {X 0,Y 239.115,Z 482.647,A -85,B 0,C 180,E1 -20131.948,E2 -20131.948} C_VEL
LIN {X 0,Y 236.716,Z 496.539,A -85,B 0,C 180,E1 -20134.265,E2 -20134.265} C_VEL
LIN {X 0,Y 234.59,Z 508.263,A -85,B 0,C 180,E1 -20136.612,E2 -20136.612} C_VEL
LIN {X 0,Y 232.49,Z 519.112,A -85,B 0,C 180,E1 -20139.194,E2 -20139.194} C_VEL
LIN {X 0,Y 230.895,Z 528.393,A -85,B 0,C 180,E1 -20141.821,E2 -20141.821} C_VEL
LIN {X 0,Y 229.32,Z 537.567,A -85,B 0,C 180,E1 -20144.9,E2 -20144.9} C_VEL
LIN {X 0,Y 228.103,Z 546.247,A -85,B 0,C 180,E1 -20148.447,E2 -20148.447} C_VEL
LIN {X 0,Y 227.311,Z 553.362,A -85,B 0,C 180,E1 -20152.056,E2 -20152.056} C_VEL
LIN {X 0,Y 227.011,Z 558.78,A -85,B 0,C 180,E1 -20155.561,E2 -20155.561} C_VEL
LIN {X 0,Y 226.892,Z 562.075,A -85,B 0,C 180,E1 -20158.225,E2 -20158.225} C_VEL
LIN {X 0,Y 227.044,Z 565.386,A -85,B 0,C 180,E1 -20161.774,E2 -20161.774} C_VEL
LIN {X 0,Y 227.927,Z 567.484,A -85,B 0,C 180,E1 -20165.307,E2 -20165.307} C_VEL
LIN {X 0,Y 229.365,Z 568.447,A -85,B 0,C 180,E1 -20168.813,E2 -20168.813} C_VEL
LIN {X 0,Y 231.301,Z 568.323,A -85,B 0,C 180,E1 -20172.28,E2 -20172.28} C_VEL
LIN {X 0,Y 234.154,Z 566.921,A -85,B 0,C 180,E1 -20176.165,E2 -20176.165} C_VEL
LIN {X 0,Y 236.913,Z 564.956,A -85,B 0,C 180,E1 -20179.045,E2 -20179.045} C_VEL
LIN {X 0,Y 242.046,Z 560.608,A -85,B 0,C 180,E1 -20183.078,E2 -20183.078} C_VEL
LIN {X 0,Y 248.425,Z 554.465,A -85,B 0,C 180,E1 -20186.913,E2 -20186.913} C_VEL
LIN {X 0,Y 255.802,Z 546.431,A -85,B 0,C 180,E1 -20190.549,E2 -20190.549} C_VEL
LIN {X 0,Y 256.58,Z 545.538,A -85,B 0,C 180,E1 -20190.894,E2 -20190.894} C_VEL
LIN {X 0,Y 258.54,Z 543.035,A -85,B 0,C 180,E1 -20192.005,E2 -20192.005} C_VEL
LIN {X 0,Y 263.238,Z 535.409,A -85,B 0,C 180,E1 -20195.876,E2 -20195.876} C_VEL
LIN {X 0,Y 265.564,Z 532.376,A -85,B 0,C 180,E1 -20196.842,E2 -20196.842} C_VEL
LIN {X 0,Y 270.085,Z 526.938,A -85,B 0,C 180,E1 -20198.132,E2 -20198.132} C_VEL
LIN {X 0,Y 270.007,Z 526.667,A -85,B 0,C 180,E1 -20198.66,E2 -20198.66} C_VEL
LIN {X 0,Y 268.971,Z 526.841,A -85,B 0,C 180,E1 -20200.786,E2 -20200.786} C_VEL
LIN {X 0,Y 267.247,Z 528.764,A -85,B 0,C 180,E1 -20202.58,E2 -20202.58} C_VEL
LIN {X 0,Y 264.831,Z 532.415,A -85,B 0,C 180,E1 -20204.789,E2 -20204.789} C_VEL
LIN {X 0,Y 261.992,Z 537.545,A -85,B 0,C 180,E1 -20207.094,E2 -20207.094} C_VEL
LIN {X 0,Y 258.832,Z 543.68,A -85,B 0,C 180,E1 -20209.333,E2 -20209.333} C_VEL
LIN {X 0,Y 255.505,Z 549.826,A -85,B 0,C 180,E1 -20211.261,E2 -20211.261} C_VEL
LIN {X 0,Y 248.287,Z 561.364,A -85,B 0,C 180,E1 -20214.53,E2 -20214.53} C_VEL
LIN {X 0,Y 243.99,Z 568.444,A -85,B 0,C 180,E1 -20216.819,E2 -20216.819} C_VEL
LIN {X 0,Y 237.345,Z 577.426,A -85,B 0,C 180,E1 -20219.776,E2 -20219.776} C_VEL
LIN {X 0,Y 232.722,Z 583.929,A -85,B 0,C 180,E1 -20222.334,E2 -20222.334} C_VEL
LIN {X 0,Y 229.715,Z 593.27,A -85,B 0,C 180,E1 -20224.639,E2 -20224.639} C_VEL
LIN {X 0,Y 226.828,Z 601.758,A -85,B 0,C 180,E1 -20227.213,E2 -20227.213} C_VEL
LIN {X 0,Y 224.302,Z 609.278,A -85,B 0,C 180,E1 -20230.049,E2 -20230.049} C_VEL
LIN {X 0,Y 222.013,Z 616.347,A -85,B 0,C 180,E1 -20233.447,E2 -20233.447} C_VEL
LIN {X 0,Y 220.115,Z 622.095,A -85,B 0,C 180,E1 -20237.085,E2 -20237.085} C_VEL
LIN {X 0,Y 219.087,Z 626.267,A -85,B 0,C 180,E1 -20240.77,E2 -20240.77} C_VEL
LIN {X 0,Y 218.595,Z 628.992,A -85,B 0,C 180,E1 -20244.465,E2 -20244.465} C_VEL
LIN {X 0,Y 218.549,Z 630.344,A -85,B 0,C 180,E1 -20248.157,E2 -20248.157} C_VEL
LIN {X 0,Y 218.609,Z 630.51,A -85,B 0,C 180,E1 -20250,E2 -20250} C_VEL
LIN {X 0,Y 218.522,Z 629.824,A -85,B 0,C 180,E1 -20253.688,E2 -20253.688} C_VEL
LIN {X 0,Y 218.788,Z 627.781,A -85,B 0,C 180,E1 -20257.382,E2 -20257.382} C_VEL
LIN {X 0,Y 219.549,Z 624.332,A -85,B 0,C 180,E1 -20261.073,E2 -20261.073} C_VEL
LIN {X 0,Y 220.918,Z 619.372,A -85,B 0,C 180,E1 -20264.744,E2 -20264.744} C_VEL
LIN {X 0,Y 222.503,Z 614.561,A -85,B 0,C 180,E1 -20267.462,E2 -20267.462} C_VEL
LIN {X 0,Y 224.741,Z 607.602,A -85,B 0,C 180,E1 -20270.598,E2 -20270.598} C_VEL
LIN {X 0,Y 227.705,Z 598.961,A -85,B 0,C 180,E1 -20273.656,E2 -20273.656} C_VEL
LIN {X 0,Y 230.676,Z 589.906,A -85,B 0,C 180,E1 -20276.217,E2 -20276.217} C_VEL
LIN {X 0,Y 233.591,Z 580.867,A -85,B 0,C 180,E1 -20278.286,E2 -20278.286} C_VEL
LIN {X 0,Y 236.732,Z 570.066,A -85,B 0,C 180,E1 -20280.311,E2 -20280.311} C_VEL
LIN {X 0,Y 238.766,Z 561.925,A -85,B 0,C 180,E1 -20281.593,E2 -20281.593} C_VEL
LIN {X 0,Y 239.038,Z 550.352,A -85,B 0,C 180,E1 -20283.454,E2 -20283.454} C_VEL
LIN {X 0,Y 238.811,Z 537.775,A -85,B 0,C 180,E1 -20285.176,E2 -20285.176} C_VEL
LIN {X 0,Y 238.105,Z 527.076,A -85,B 0,C 180,E1 -20286.455,E2 -20286.455} C_VEL
LIN {X 0,Y 235.43,Z 513.975,A -85,B 0,C 180,E1 -20288.03,E2 -20288.03} C_VEL
LIN {X 0,Y 231.22,Z 500.253,A -85,B 0,C 180,E1 -20289.622,E2 -20289.622} C_VEL
LIN {X 0,Y 227.521,Z 490.435,A -85,B 0,C 180,E1 -20290.815,E2 -20290.815} C_VEL
LIN {X 0,Y 226.546,Z 477.165,A -85,B 0,C 180,E1 -20295.04,E2 -20295.04} C_VEL
LIN {X 0,Y 225.616,Z 468.888,A -85,B 0,C 180,E1 -20297.955,E2 -20297.955} C_VEL
LIN {X 0,Y 224.708,Z 463.396,A -85,B 0,C 180,E1 -20300.122,E2 -20300.122} C_VEL
LIN {X 0,Y 222.381,Z 454.69,A -85,B 0,C 180,E1 -20304.499,E2 -20304.499} C_VEL
LIN {X 0,Y 221.501,Z 449.397,A -85,B 0,C 180,E1 -20309.492,E2 -20309.492} C_VEL
LIN {X 0,Y 220.988,Z 446.57,A -85,B 0,C 180,E1 -20312.329,E2 -20312.329} C_VEL
LIN {X 0,Y 220.879,Z 446.585,A -85,B 0,C 180,E1 -20317.554,E2 -20317.554} C_VEL
LIN {X 0,Y 220.986,Z 446.583,A -85,B 0,C 180,E1 -20322.571,E2 -20322.571} C_VEL
LIN {X 0,Y 221.013,Z 446.569,A -85,B 0,C 180,E1 -20327.139,E2 -20327.139} C_VEL
LIN {X 0,Y 221.202,Z 446.529,A -85,B 0,C 180,E1 -20330.859,E2 -20330.859} C_VEL
LIN {X 0,Y 221.139,Z 446.563,A -85,B 0,C 180,E1 -20334.529,E2 -20334.529} C_VEL
LIN {X 0,Y 221.514,Z 446.495,A -85,B 0,C 180,E1 -20338.182,E2 -20338.182} C_VEL
LIN {X 0,Y 221.514,Z 446.497,A -85,B 0,C 180,E1 -20341.818,E2 -20341.818} C_VEL
LIN {X 0,Y 221.292,Z 446.528,A -85,B 0,C 180,E1 -20347.298,E2 -20347.298} C_VEL
LIN {X 0,Y 221.114,Z 446.567,A -85,B 0,C 180,E1 -20350.994,E2 -20350.994} C_VEL
LIN {X 0,Y 221.018,Z 446.579,A -85,B 0,C 180,E1 -20356.63,E2 -20356.63} C_VEL
LIN {X 0,Y 220.943,Z 446.716,A -85,B 0,C 180,E1 -20358.376,E2 -20358.376} C_VEL
LIN {X 0,Y 222.803,Z 452.385,A -85,B 0,C 180,E1 -20363.828,E2 -20363.828} C_VEL
LIN {X 0,Y 224.308,Z 457.337,A -85,B 0,C 180,E1 -20368.033,E2 -20368.033} C_VEL
LIN {X 0,Y 225.672,Z 462.471,A -85,B 0,C 180,E1 -20371.967,E2 -20371.967} C_VEL
LIN {X 0,Y 227.095,Z 468.8,A -85,B 0,C 180,E1 -20376.425,E2 -20376.425} C_VEL
LIN {X 0,Y 228.208,Z 474.796,A -85,B 0,C 180,E1 -20380.295,E2 -20380.295} C_VEL
LIN {X 0,Y 229.092,Z 480.303,A -85,B 0,C 180,E1 -20383.65,E2 -20383.65} C_VEL
LIN {X 0,Y 229.76,Z 485.185,A -85,B 0,C 180,E1 -20386.441,E2 -20386.441} C_VEL
LIN {X 0,Y 229.671,Z 487.585,A -85,B 0,C 180,E1 -20387.685,E2 -20387.685} C_VEL
LIN {X 0,Y 229.04,Z 491.364,A -85,B 0,C 180,E1 -20389.47,E2 -20389.47} C_VEL
LIN {X 0,Y 234.093,Z 506.373,A -85,B 0,C 180,E1 -20391.231,E2 -20391.231} C_VEL
LIN {X 0,Y 237.285,Z 518.709,A -85,B 0,C 180,E1 -20392.754,E2 -20392.754} C_VEL
LIN {X 0,Y 239.29,Z 530.045,A -85,B 0,C 180,E1 -20394.228,E2 -20394.228} C_VEL
LIN {X 0,Y 240.633,Z 542.523,A -85,B 0,C 180,E1 -20396.01,E2 -20396.01} C_VEL
LIN {X 0,Y 240.912,Z 552.59,A -85,B 0,C 180,E1 -20397.586,E2 -20397.586} C_VEL
LIN {X 0,Y 237.897,Z 565.129,A -85,B 0,C 180,E1 -20399.43,E2 -20399.43} C_VEL
LIN {X 0,Y 234.722,Z 575.847,A -85,B 0,C 180,E1 -20401.375,E2 -20401.375} C_VEL
LIN {X 0,Y 231.234,Z 586.692,A -85,B 0,C 180,E1 -20403.851,E2 -20403.851} C_VEL
LIN {X 0,Y 228.211,Z 595.642,A -85,B 0,C 180,E1 -20406.4,E2 -20406.4} C_VEL
LIN {X 0,Y 225.048,Z 604.426,A -85,B 0,C 180,E1 -20409.533,E2 -20409.533} C_VEL
LIN {X 0,Y 223.002,Z 611.079,A -85,B 0,C 180,E1 -20412.579,E2 -20412.579} C_VEL
LIN {X 0,Y 220.814,Z 617.253,A -85,B 0,C 180,E1 -20416.19,E2 -20416.19} C_VEL
LIN {X 0,Y 219.749,Z 620.761,A -85,B 0,C 180,E1 -20418.937,E2 -20418.937} C_VEL
LIN {X 0,Y 218.869,Z 624.182,A -85,B 0,C 180,E1 -20422.62,E2 -20422.62} C_VEL
LIN {X 0,Y 218.519,Z 626.212,A -85,B 0,C 180,E1 -20426.312,E2 -20426.312} C_VEL
LIN {X 0,Y 218.536,Z 626.905,A -85,B 0,C 180,E1 -20430,E2 -20430} C_VEL
LIN {X 0,Y 218.514,Z 626.265,A -85,B 0,C 180,E1 -20433.688,E2 -20433.688} C_VEL
LIN {X 0,Y 218.868,Z 624.278,A -85,B 0,C 180,E1 -20437.38,E2 -20437.38} C_VEL
LIN {X 0,Y 219.739,Z 620.906,A -85,B 0,C 180,E1 -20441.064,E2 -20441.064} C_VEL
LIN {X 0,Y 221.154,Z 616.045,A -85,B 0,C 180,E1 -20444.728,E2 -20444.728} C_VEL
LIN {X 0,Y 222.942,Z 611.329,A -85,B 0,C 180,E1 -20447.426,E2 -20447.426} C_VEL
LIN {X 0,Y 225.277,Z 604.319,A -85,B 0,C 180,E1 -20450.623,E2 -20450.623} C_VEL
LIN {X 0,Y 228.136,Z 596.011,A -85,B 0,C 180,E1 -20453.608,E2 -20453.608} C_VEL
LIN {X 0,Y 231.15,Z 587.133,A -85,B 0,C 180,E1 -20456.159,E2 -20456.159} C_VEL
LIN {X 0,Y 234.621,Z 576.382,A -85,B 0,C 180,E1 -20458.638,E2 -20458.638} C_VEL
LIN {X 0,Y 237.707,Z 566.066,A -85,B 0,C 180,E1 -20460.536,E2 -20460.536} C_VEL
LIN {X 0,Y 240.519,Z 554.888,A -85,B 0,C 180,E1 -20462.226,E2 -20462.226} C_VEL
LIN {X 0,Y 241.043,Z 551.878,A -85,B 0,C 180,E1 -20462.643,E2 -20462.643} C_VEL
LIN {X 0,Y 240.518,Z 540.322,A -85,B 0,C 180,E1 -20464.438,E2 -20464.438} C_VEL
LIN {X 0,Y 238.948,Z 527.362,A -85,B 0,C 180,E1 -20466.253,E2 -20466.253} C_VEL
LIN {X 0,Y 236.325,Z 514.365,A -85,B 0,C 180,E1 -20467.923,E2 -20467.923} C_VEL
LIN {X 0,Y 232.532,Z 501.262,A -85,B 0,C 180,E1 -20469.513,E2 -20469.513} C_VEL
LIN {X 0,Y 229.077,Z 491.276,A -85,B 0,C 180,E1 -20470.705,E2 -20470.705} C_VEL
LIN {X 0,Y 229.796,Z 486.977,A -85,B 0,C 180,E1 -20472.776,E2 -20472.776} C_VEL
LIN {X 0,Y 229.488,Z 482.517,A -85,B 0,C 180,E1 -20475.221,E2 -20475.221} C_VEL
LIN {X 0,Y 228.61,Z 476.821,A -85,B 0,C 180,E1 -20478.626,E2 -20478.626} C_VEL
LIN {X 0,Y 227.41,Z 470.017,A -85,B 0,C 180,E1 -20482.942,E2 -20482.942} C_VEL
LIN {X 0,Y 225.876,Z 463.349,A -85,B 0,C 180,E1 -20487.583,E2 -20487.583} C_VEL
LIN {X 0,Y 225.822,Z 462.92,A -85,B 0,C 180,E1 -20488.001,E2 -20488.001} C_VEL
LIN {X 0,Y 227.393,Z 467.332,A -85,B 0,C 180,E1 -20488.735,E2 -20488.735} C_VEL
LIN {X 0,Y 231.473,Z 481.297,A -85,B 0,C 180,E1 -20491.153,E2 -20491.153} C_VEL
LIN {X 0,Y 232.038,Z 484.295,A -85,B 0,C 180,E1 -20491.699,E2 -20491.699} C_VEL
LIN {X 0,Y 229.782,Z 497.091,A -85,B 0,C 180,E1 -20493.917,E2 -20493.917} C_VEL
LIN {X 0,Y 227.594,Z 508.783,A -85,B 0,C 180,E1 -20496.332,E2 -20496.332} C_VEL
LIN {X 0,Y 225.237,Z 520.773,A -85,B 0,C 180,E1 -20499.294,E2 -20499.294} C_VEL
LIN {X 0,Y 223.641,Z 530.409,A -85,B 0,C 180,E1 -20502.158,E2 -20502.158} C_VEL
LIN {X 0,Y 222.049,Z 539.413,A -85,B 0,C 180,E1 -20505.333,E2 -20505.333} C_VEL
LIN {X 0,Y 221.106,Z 545.957,A -85,B 0,C 180,E1 -20508.076,E2 -20508.076} C_VEL
LIN {X 0,Y 220.321,Z 552.644,A -85,B 0,C 180,E1 -20511.443,E2 -20511.443} C_VEL
LIN {X 0,Y 220.013,Z 557.619,A -85,B 0,C 180,E1 -20514.501,E2 -20514.501} C_VEL
LIN {X 0,Y 219.8,Z 562.364,A -85,B 0,C 180,E1 -20518.168,E2 -20518.168} C_VEL
LIN {X 0,Y 219.985,Z 565.847,A -85,B 0,C 180,E1 -20521.831,E2 -20521.831} C_VEL
LIN {X 0,Y 220.895,Z 568.166,A -85,B 0,C 180,E1 -20525.477,E2 -20525.477} C_VEL
LIN {X 0,Y 222.432,Z 569.355,A -85,B 0,C 180,E1 -20529.09,E2 -20529.09} C_VEL
LIN {X 0,Y 224.475,Z 569.478,A -85,B 0,C 180,E1 -20532.66,E2 -20532.66} C_VEL
LIN {X 0,Y 227.741,Z 568.217,A -85,B 0,C 180,E1 -20536.932,E2 -20536.932} C_VEL
LIN {X 0,Y 230.415,Z 566.629,A -85,B 0,C 180,E1 -20539.604,E2 -20539.604} C_VEL
LIN {X 0,Y 234.679,Z 563.554,A -85,B 0,C 180,E1 -20542.912,E2 -20542.912} C_VEL
LIN {X 0,Y 238.366,Z 560.548,A -85,B 0,C 180,E1 -20545.31,E2 -20545.31} C_VEL
LIN {X 0,Y 243.971,Z 555.528,A -85,B 0,C 180,E1 -20548.38,E2 -20548.38} C_VEL
LIN {X 0,Y 251.411,Z 548.137,A -85,B 0,C 180,E1 -20551.818,E2 -20551.818} C_VEL
LIN {X 0,Y 259.058,Z 539.914,A -85,B 0,C 180,E1 -20554.73,E2 -20554.73} C_VEL
LIN {X 0,Y 265.564,Z 532.376,A -85,B 0,C 180,E1 -20556.842,E2 -20556.842} C_VEL
LIN {X 0,Y 266.381,Z 531.284,A -85,B 0,C 180,E1 -20557.286,E2 -20557.286} C_VEL
LIN {X 0,Y 266.574,Z 530.611,A -85,B 0,C 180,E1 -20558.098,E2 -20558.098} C_VEL
LIN {X 0,Y 265.975,Z 530.803,A -85,B 0,C 180,E1 -20558.942,E2 -20558.942} C_VEL
LIN {X 0,Y 263.168,Z 532.972,A -85,B 0,C 180,E1 -20561.427,E2 -20561.427} C_VEL
LIN {X 0,Y 262.248,Z 534,A -85,B 0,C 180,E1 -20562.347,E2 -20562.347} C_VEL
LIN {X 0,Y 259.252,Z 538.166,A -85,B 0,C 180,E1 -20564.816,E2 -20564.816} C_VEL
LIN {X 0,Y 255.906,Z 543.517,A -85,B 0,C 180,E1 -20567.179,E2 -20567.179} C_VEL
LIN {X 0,Y 252.674,Z 548.865,A -85,B 0,C 180,E1 -20569.138,E2 -20569.138} C_VEL
LIN {X 0,Y 248.78,Z 554.886,A -85,B 0,C 180,E1 -20571.056,E2 -20571.056} C_VEL
LIN {X 0,Y 240.324,Z 566.896,A -85,B 0,C 180,E1 -20574.799,E2 -20574.799} C_VEL
LIN {X 0,Y 237.186,Z 571.258,A -85,B 0,C 180,E1 -20576.293,E2 -20576.293} C_VEL
LIN {X 0,Y 229.81,Z 580.435,A -85,B 0,C 180,E1 -20579.695,E2 -20579.695} C_VEL
LIN {X 0,Y 225.842,Z 585.668,A -85,B 0,C 180,E1 -20581.922,E2 -20581.922} C_VEL
LIN {X 0,Y 222.74,Z 594.711,A -85,B 0,C 180,E1 -20584.288,E2 -20584.288} C_VEL
LIN {X 0,Y 219.79,Z 602.94,A -85,B 0,C 180,E1 -20586.939,E2 -20586.939} C_VEL
LIN {X 0,Y 217.157,Z 610.544,A -85,B 0,C 180,E1 -20590.011,E2 -20590.011} C_VEL
LIN {X 0,Y 215.167,Z 616.291,A -85,B 0,C 180,E1 -20592.904,E2 -20592.904} C_VEL
LIN {X 0,Y 213.15,Z 622.038,A -85,B 0,C 180,E1 -20596.656,E2 -20596.656} C_VEL
LIN {X 0,Y 212.057,Z 626.209,A -85,B 0,C 180,E1 -20600.462,E2 -20600.462} C_VEL
LIN {X 0,Y 211.508,Z 628.934,A -85,B 0,C 180,E1 -20604.279,E2 -20604.279} C_VEL
LIN {X 0,Y 211.45,Z 630.285,A -85,B 0,C 180,E1 -20608.095,E2 -20608.095} C_VEL
LIN {X 0,Y 211.508,Z 630.452,A -85,B 0,C 180,E1 -20610,E2 -20610} C_VEL
LIN {X 0,Y 211.436,Z 629.765,A -85,B 0,C 180,E1 -20613.812,E2 -20613.812} C_VEL
LIN {X 0,Y 211.712,Z 627.722,A -85,B 0,C 180,E1 -20617.631,E2 -20617.631} C_VEL
LIN {X 0,Y 212.53,Z 624.273,A -85,B 0,C 180,E1 -20621.444,E2 -20621.444} C_VEL
LIN {X 0,Y 214.038,Z 619.313,A -85,B 0,C 180,E1 -20625.229,E2 -20625.229} C_VEL
LIN {X 0,Y 215.687,Z 614.503,A -85,B 0,C 180,E1 -20628.032,E2 -20628.032} C_VEL
LIN {X 0,Y 218.057,Z 607.544,A -85,B 0,C 180,E1 -20631.259,E2 -20631.259} C_VEL
LIN {X 0,Y 221.173,Z 598.904,A -85,B 0,C 180,E1 -20634.399,E2 -20634.399} C_VEL
LIN {X 0,Y 224.283,Z 589.851,A -85,B 0,C 180,E1 -20637.024,E2 -20637.024} C_VEL
LIN {X 0,Y 228.009,Z 578.855,A -85,B 0,C 180,E1 -20639.549,E2 -20639.549} C_VEL
LIN {X 0,Y 231.204,Z 567.757,A -85,B 0,C 180,E1 -20641.594,E2 -20641.594} C_VEL
LIN {X 0,Y 232.512,Z 562.105,A -85,B 0,C 180,E1 -20642.504,E2 -20642.504} C_VEL
LIN {X 0,Y 232.891,Z 549.72,A -85,B 0,C 180,E1 -20644.547,E2 -20644.547} C_VEL
LIN {X 0,Y 232.739,Z 536.159,A -85,B 0,C 180,E1 -20646.426,E2 -20646.426} C_VEL
LIN {X 0,Y 232.228,Z 528.969,A -85,B 0,C 180,E1 -20647.33,E2 -20647.33} C_VEL
LIN {X 0,Y 229.831,Z 516.411,A -85,B 0,C 180,E1 -20648.938,E2 -20648.938} C_VEL
LIN {X 0,Y 226.176,Z 503.722,A -85,B 0,C 180,E1 -20650.517,E2 -20650.517} C_VEL
LIN {X 0,Y 221.196,Z 490.444,A -85,B 0,C 180,E1 -20652.255,E2 -20652.255} C_VEL
LIN {X 0,Y 220.546,Z 478.965,A -85,B 0,C 180,E1 -20656.125,E2 -20656.125} C_VEL
LIN {X 0,Y 219.926,Z 472.629,A -85,B 0,C 180,E1 -20658.464,E2 -20658.464} C_VEL
LIN {X 0,Y 219.327,Z 468.212,A -85,B 0,C 180,E1 -20660.268,E2 -20660.268} C_VEL
LIN {X 0,Y 217.192,Z 460.026,A -85,B 0,C 180,E1 -20664.377,E2 -20664.377} C_VEL
LIN {X 0,Y 214.506,Z 450.375,A -85,B 0,C 180,E1 -20670.564,E2 -20670.564} C_VEL
LIN {X 0,Y 213.898,Z 447.445,A -85,B 0,C 180,E1 -20673.01,E2 -20673.01} C_VEL
LIN {X 0,Y 213.854,Z 447.47,A -85,B 0,C 180,E1 -20676.953,E2 -20676.953} C_VEL
LIN {X 0,Y 213.945,Z 447.455,A -85,B 0,C 180,E1 -20682.804,E2 -20682.804} C_VEL
LIN {X 0,Y 213.954,Z 447.441,A -85,B 0,C 180,E1 -20686.707,E2 -20686.707} C_VEL
LIN {X 0,Y 214.14,Z 447.409,A -85,B 0,C 180,E1 -20690.555,E2 -20690.555} C_VEL
LIN {X 0,Y 214.1,Z 447.442,A -85,B 0,C 180,E1 -20694.349,E2 -20694.349} C_VEL
LIN {X 0,Y 214.447,Z 447.374,A -85,B 0,C 180,E1 -20698.122,E2 -20698.122} C_VEL
LIN {X 0,Y 214.557,Z 447.385,A -85,B 0,C 180,E1 -20700,E2 -20700} C_VEL
LIN {X 0,Y 214.447,Z 447.376,A -85,B 0,C 180,E1 -20701.878,E2 -20701.878} C_VEL
LIN {X 0,Y 214.23,Z 447.405,A -85,B 0,C 180,E1 -20707.54,E2 -20707.54} C_VEL
LIN {X 0,Y 214.047,Z 447.45,A -85,B 0,C 180,E1 -20711.362,E2 -20711.362} C_VEL
LIN {X 0,Y 213.953,Z 447.445,A -85,B 0,C 180,E1 -20714.749,E2 -20714.749} C_VEL
LIN {X 0,Y 215.165,Z 451.342,A -85,B 0,C 180,E1 -20719.065,E2 -20719.065} C_VEL
LIN {X 0,Y 216.731,Z 456.14,A -85,B 0,C 180,E1 -20723.931,E2 -20723.931} C_VEL
LIN {X 0,Y 218.107,Z 460.683,A -85,B 0,C 180,E1 -20727.855,E2 -20727.855} C_VEL
LIN {X 0,Y 219.383,Z 465.738,A -85,B 0,C 180,E1 -20731.91,E2 -20731.91} C_VEL
LIN {X 0,Y 220.634,Z 471.552,A -85,B 0,C 180,E1 -20736.107,E2 -20736.107} C_VEL
LIN {X 0,Y 221.521,Z 476.425,A -85,B 0,C 180,E1 -20739.385,E2 -20739.385} C_VEL
LIN {X 0,Y 222.562,Z 482.91,A -85,B 0,C 180,E1 -20743.424,E2 -20743.424} C_VEL
LIN {X 0,Y 223.186,Z 488.02,A -85,B 0,C 180,E1 -20746.407,E2 -20746.407} C_VEL
LIN {X 0,Y 222.796,Z 491.401,A -85,B 0,C 180,E1 -20748.086,E2 -20748.086} C_VEL
LIN {X 0,Y 228.001,Z 506.812,A -85,B 0,C 180,E1 -20750.02,E2 -20750.02} C_VEL
LIN {X 0,Y 231.39,Z 520.194,A -85,B 0,C 180,E1 -20751.774,E2 -20751.774} C_VEL
LIN {X 0,Y 233.437,Z 532.722,A -85,B 0,C 180,E1 -20753.508,E2 -20753.508} C_VEL
LIN {X 0,Y 234.515,Z 544.518,A -85,B 0,C 180,E1 -20755.292,E2 -20755.292} C_VEL
LIN {X 0,Y 234.618,Z 554.164,A -85,B 0,C 180,E1 -20756.86,E2 -20756.86} C_VEL
LIN {X 0,Y 231.768,Z 565.341,A -85,B 0,C 180,E1 -20758.564,E2 -20758.564} C_VEL
LIN {X 0,Y 228.521,Z 575.9,A -85,B 0,C 180,E1 -20760.523,E2 -20760.523} C_VEL
LIN {X 0,Y 224.871,Z 586.748,A -85,B 0,C 180,E1 -20763.052,E2 -20763.052} C_VEL
LIN {X 0,Y 221.696,Z 595.699,A -85,B 0,C 180,E1 -20765.662,E2 -20765.662} C_VEL
LIN {X 0,Y 218.813,Z 603.369,A -85,B 0,C 180,E1 -20768.422,E2 -20768.422} C_VEL
LIN {X 0,Y 216.843,Z 609.352,A -85,B 0,C 180,E1 -20771.089,E2 -20771.089} C_VEL
LIN {X 0,Y 214.923,Z 614.438,A -85,B 0,C 180,E1 -20773.862,E2 -20773.862} C_VEL
LIN {X 0,Y 213.102,Z 619.767,A -85,B 0,C 180,E1 -20777.622,E2 -20777.622} C_VEL
LIN {X 0,Y 212.244,Z 622.71,A -85,B 0,C 180,E1 -20780.47,E2 -20780.47} C_VEL
LIN {X 0,Y 211.577,Z 625.425,A -85,B 0,C 180,E1 -20784.281,E2 -20784.281} C_VEL
LIN {X 0,Y 211.397,Z 626.783,A -85,B 0,C 180,E1 -20788.095,E2 -20788.095} C_VEL
